// Types/States/MurrIOMOdule/MOM_STATES
{attribute 'strict'}
{attribute 'qualified_only'}
TYPE MOM_STATES :
(
	Idle := 0,
	Reverse := 1,
	Reversing := 2,
	ReverseToPrinthead := 3,
	ReversingToPrintHead := 4,
	ReverseDone := 5,
	WaitingForPrinter := 10,
	FeedToPrintOffset := 11,
	FeedingToPrintOffset := 12,
	FedToPrintOffset := 13,
	FeedAtPrintSpeed := 20,
	FeedingAtPrintSpeed := 21,
	FedAtPrintSpeed := 22,
	FeedBagOut := 30,
	FeedingBagOut := 31,
	FedBagOut := 32,
	Ready := 40,
	FeedToEye := 50,
	FeedingToEye := 51,
	SetTorqueMode := 52,
	Fault := 99,
	Manual := 100
);
END_TYPE

// Types/States/JOG_STATES
{attribute 'strict'}
{attribute 'qualified_only'}
TYPE JOG_STATES :
(
    Idle := 0,
    JogForwardDIRequest := 10,
    JogForwardOpcodeRequest := 11,
    JoggingForward := 12,
    JogReverseDIRequest := 20,
    JogReverseOpcodeRequest := 21,
    JoggingReverse := 22,
    StoppingJog := 30
);
END_TYPE

// Types/Fault
TYPE Fault :
STRUCT
    name : STRING[20];
    description : STRING[255];
END_STRUCT
END_TYPE

// Types/QX_PROGRAMS
{attribute 'strict'}
TYPE QX_PROGRAMS :
(
    HOME_HARD_STOP := 1
);
END_TYPE

// Types/Factoy Selection/ExteralConveyorSelection
{attribute 'qualified_only'}
{attribute 'strict'}
TYPE ExteralConveyorSelection :
(
	NotInstalled := 0,
	ExternalExitConveyor := 1
);
END_TYPE

// Types/PRINT_SPEEDS
{attribute 'qualified_only'}
{attribute 'strict'}
TYPE PRINT_SPEEDS :
(
	Two_IPS := 2
);
END_TYPE

// Types/States/PRESSURE_BAR_STATES
{attribute 'strict'}
{attribute 'qualified_only'}
TYPE PRESSURE_BAR_STATES :
(
	Idle := 0,
	OpenJaw := 10,
	OpeningJaw := 11,
	JawOpened := 12,
	CloseJaw := 20,
	ClosingJaw := 21,
	JawClosed := 22,
	Sealing := 30,
	Manual := 40,
	Homing := 41,
	Fault := 99
);
END_TYPE

// Types/Factoy Selection/BCVSelection
{attribute 'qualified_only'}
{attribute 'strict'}
TYPE BCVSelection :
(
	NotInstalled := 0,
	VisionBased := 1,
	LaserScanner := 2,
	TwoDimensional := 3
);
END_TYPE

// Types/States/MurrIOMOdule/MURR_SYSTEM_STATES
{attribute 'qualified_only'}
TYPE MURR_SYSTEM_STATES :
(
	Internal_Comm_OK := 1,
	Waiting_For_MOM := 2,
	Configuring_MOM := 4,
	Internal_Comm_Disabled := 8,
	No_Comm_To_Configured_Node := 127
);
END_TYPE

// Types/States/Head/HEAD_STATES
{attribute 'qualified_only'}
{attribute 'strict'}
TYPE HEAD_STATES :
(
	Idle := 0,
	SealAndSeparateBag := 10,
	SealingAndSeparatingBag := 11,
	SealedAndSeparatedBag := 12,
	ReleaseAndFeedBag := 20,
	ReleasingAndFeedingBag := 21,
	ReleasedAndFedBag := 22,
	OpenBag := 30,
	OpeningBag := 31,
	OpenedBag := 32,
	FinishCycle := 40, 
	FinishingCycle := 41,
	FinishedCycle := 42,
	StartReset := 50,
	Resetting := 51,
	StartHoming := 53,
	Homing := 54,
	HomingComplete := 55,
	MovePassthrough := 60,
	MovingPassthrough := 61,
	MovedPassthrough := 62,
	Fault := 99
);
END_TYPE

// Types/States/Head/SEAL_FLATTENER_STATES
{attribute 'strict'}
{attribute 'qualified_only'}
TYPE SEAL_FLATTENER_STATES :
(
	Idle := 0,
	MoveFlattenersOut := 10,
	MovingFlattenersOut := 11,
	MovedFlattenersOut := 12,
	MoveFlattenersUpAndToClearance := 20,
	MovingFlattenersUpAndToClearance := 21,
	MovedFlattenersUpAndToClearance := 22,
	MoveFlattenersToBagFeed := 23,
	MovingFlattenersToBagFeed := 24,
	MovedFlattenersToBagFeed := 25,
	MoveFlattenersIn := 30,
	MovingFlattenersIn := 31,
	MovedFlattenersIn := 32,
	MoveFlattenersDown := 40,
	MovingFlattenersDown := 41,
	MovedFlattenersDown := 42,
	MoveFlattenersToBagHolding := 50,
	MovingFlattenersToBagHolding := 51,
	MovedFlattenersToBagHolding := 52,
	Ready := 60,
	Fault := 99
);
END_TYPE

// Types/Factoy Selection/BagDeflatorSelection
{attribute 'qualified_only'}
{attribute 'strict'}
TYPE BagDeflatorSelection :
(
	NotInstalled := 0,
	IBDStandard := 1,
	IBDWithHingedPlate := 2,
	MotorizedIBD := 3
);
END_TYPE

// Types/States/Head/SEAL_BAR_STATES
{attribute 'strict'}
{attribute 'qualified_only'}
TYPE SEAL_BAR_STATES :
(
	Idle := 0,
	ExtendSealBar := 10,
	ExtendingSealBar := 11,
	SealBarExtened := 12,
	RetractSealBar := 20,
	RetractingSealBar := 21,
	RetractedSealBar := 22,
	Fault := 99
);
END_TYPE

// Types/States/Head/SEAL_SEPARATE_STATES
{attribute 'qualified_only'}
{attribute 'strict'}
TYPE SEAL_SEPARATE_STATES :
(
	Idle := 0,
	BringInIBD := 8,
	WaitForJawCloseDelay := 9,
	MoveJawIn := 10,
	MovingJawIn := 11,
	MovedJawIn := 12,
	ReverseBag := 20,
	ReversingBag := 21,
	ReversedBag := 22,
	SealBag := 30, 
	SealingBag := 31, 
	SealedBag := 32,
	Done := 100,
	Fault := 99
);
END_TYPE

// Types/ServiceCommands
TYPE ServiceCommands : 
STRUCT
	extendCommand : BOOL;
	retractCommand : BOOL;
	exhaustCommand : BOOL;
	extendedFeedback : BOOL;
	retractedFeedback : BOOL;
END_STRUCT
END_TYPE

// Types/States/VACUUM_PICKER_STATES
{attribute 'strict'}
{attribute 'qualified_only'}
TYPE VACUUM_PICKER_STATES :
(
	Idle := 0,
	Home := 1, 
	Homing := 2, 
	Homed := 3,
	XAxisMoveIn := 10,
	XAxisMovingIn := 11, 
	XaxisMovedIn := 12,
	VacuumTurnOn := 20,
	VacuumHeadDown := 30,
	YAxisMoveDown := 31,
	VacuumHeadAndYAxisMovingDown := 32,
	VacuumHeadAndYAxisMovedDown := 33,
	VacuumTurnOff := 40,
	ConveyorTurnOn := 50,
	ConveyorMoving := 51,
	ConveyorDone := 52,

	Fault := 99,
	Ready := 100,
	Manual := 101
);
END_TYPE

// FBs/Components/FB_MotorizedIBD/MotorizedIBDStates
{attribute 'qualified_only'}
{attribute 'strict'}
TYPE MotorizedIBDStates :
(
	Idle := 0,
	Homing := 9,
	Initialize := 10,
	Initializing := 11,
	Initialized := 12,
	MoveJawOut := 20,
	MovingJawOut := 21,
	MovedJawOut := 22,
	MoveJawIn := 30,
	MovingJawIn := 31,
	MovedJawIn := 32,
	StartClamping := 40,
	StartedClamping := 41,
	Clamping := 42, 
	ReleaseClamp := 43, 
	ReleasingClamp := 44,
	MoveOutFull := 50,
	MovingOutFull := 51,
	MovedOutFull := 52,
	Faulting := 98,
	Faulted := 99
);
END_TYPE

// FBs/Components/DelayDwellFB/DELAY_DWELL_STATES
{attribute 'qualified_only'}
{attribute 'strict'}
TYPE DELAY_DWELL_STATES :
(
	Idle := 0,
	Delay := 1,
	Dwell := 2,
	ResettingDwell := 10,
	ManualOn := 20,
	ManualOff := 21
);
END_TYPE

// Types/Factoy Selection/SealFlattenerSelection
{attribute 'qualified_only'}
{attribute 'strict'}
TYPE SealFlattenerSelection :
(
	NotInstalled := 0,
	MotorizedSealFlatteners := 1
);
END_TYPE

// Types/States/OPCODE_MODBUS_COMMAND_STATES
{attribute 'strict'}
{attribute 'qualified_only'}
TYPE OPCODE_MODBUS_COMMAND_STATES :
(
	Idle := 0,
	SendOpcodeAndParameters := 10,
	WaitAfterOpcodeAndParametersSent := 11,
	Fault := 99
);
END_TYPE

// Types/States/FILLER_STATES
{attribute 'strict'}
{attribute 'qualified_only'}
TYPE FILLER_STATES :
(
	Idle := 0,
	CycleBaggerToActiveFiller := 10,
	WaitingForFiller := 11,
	Dropping := 13,
	BaggerCycling := 14,
	Fault := 99
);
END_TYPE

// Types/States/Head/FINISH_CYCLE_STATES
{attribute 'qualified_only'}
{attribute 'strict'}
TYPE FINISH_CYCLE_STATES :
(
	Idle := 0,
	Start := 1,
	OpenFunnel := 10, 
	OpeningFunnel := 11, 
	OpenedFunnel := 12,
	ClosingFunnelForRetry := 13,
	FunnelClosed := 14,
	BringSealFlattenersInAndDown := 20, 
	BringingSealFlattenersInAndDown := 21,
	SealFlattenersInAndDown := 22,
	BringSealFlattenersToBagHolding := 30,
	BringingSealFlattenersToBagHolding := 31,
	SealFlattenersAtBagHolding := 32,
	Done := 100,
	Fault := 99
);
END_TYPE

// Types/States/GRABBER_STATES
{attribute 'strict'}
{attribute 'qualified_only'}
TYPE GRABBER_STATES :
(
	Idle := 0,
	OpenGrippers := 10,
	MoveGrippersOut := 11,
	MovingGrippersOut := 12,
	GrippersMovedOut :=13,
	MoveGantryUp := 20,
	MovingGantryUp := 21,
	GantryMovedUp := 22,
	MoveGrippersIn := 30,
	MovingGrippersIn := 31,
	GrippersMovedIn := 32,
	Ready := 40,
	GrabBag := 50,
	MoveGantryDown := 60,
	MovingGantryDown := 61,
	GantryMovedDown := 62,
	ReleaseBag := 70,
	Fault := 99
);
END_TYPE

// Types/Factoy Selection/PalmButtonSelection
{attribute 'qualified_only'}
{attribute 'strict'}
TYPE PalmButtonSelection :
(
	NotInstalled := 0,
	SinglePalmButton := 1,
	DualPalmButton := 2,
	LightedPalmButton := 3
);
END_TYPE

// FBs/Fault/LogMessageType
TYPE LogMessageType :
STRUCT
	logTime : DATE_AND_TIME;
	logMessage : STRING;
END_STRUCT
END_TYPE

// Types/ORIENTAL_OPERATION_TYPES
{attribute 'qualified_only'}
{attribute 'strict'}
TYPE ORIENTAL_OPERATION_TYPES :
(
    NoSetting := 0,
    AbsolutePositioning := 1,
    IncrementalPositioning := 2
);
END_TYPE

// FBs/Components/KeyenceL20FB/eKeyenceLN20_Error_ID
{attribute 'qualified_only'}
{attribute 'strict'}
TYPE eKeyenceLN20_Error_ID :
(
	NO_ERROR := 0,
	OPERATION_INSTRUCTION_ERROR := 120,
	BANK_NUMBER_ERROR := 102,
	EIP_UPDATE_ERROR := 230
);
END_TYPE

// FBs/Components/FB_MotorizedPressureBar/MotorizedPbarStates
{attribute 'qualified_only'}
{attribute 'strict'}
TYPE MotorizedPbarStates :
(
	Idle := 0,
	Homing := 9,
	Initialize := 10,
	Initializing := 11,
	Initialized := 12,
	MoveJawOut := 20,
	MovingJawOut := 21,
	MovedJawOut := 22,
	MoveJawIn := 30,
	MovingJawIn := 31,
	MovedJawIn := 32,
	StartClamping := 40,
	StartedClamping := 41,
	Clamping := 42, 
	ReleaseClamp := 43, 
	ReleasingClamp := 44,
	Faulting := 98,
	Faulted := 99
);
END_TYPE

// Types/States/BCR_STATES
{attribute 'strict'}
{attribute 'qualified_only'}
TYPE BCR_STATES :
(
	Idle := 0,
	WaitForOffset := 10,
	TriggerReader := 11,
	WaitingForResult := 12,
	Resetting := 13
);
END_TYPE

// Types/PressureBarFaultsType
TYPE PressureBarFaultsType :
STRUCT
	failedToOpen : FB_Fault(name := 'Pressure Bar Failed to Open');        // Pressure Bar was commanded to extend but failed to reach the sensor
    failedToClose : FB_Fault(name := 'Pressure Bar Failed to Close');      // Pressure Bar was commanded to retract but failed to reach the sensor
	sensorFault : FB_Fault(name := 'Pressure Bar Sensor Fault');		// Both the open and close sensors active at the same time
	obstructionDetected : FB_Fault(name := 'Pressure Bar Obstruction Detected');		// Pressure Bar detected an obstruction
	obstructionFailedToSwitch : FB_Fault(name := 'Pressure Bar Obstruction Detected'); // Pressure bar obstruction sensors should switch when closed
END_STRUCT
END_TYPE

// Types/Factoy Selection/BagOpenFingersSelection
{attribute 'qualified_only'}
{attribute 'strict'}
TYPE BagOpenFingersSelection :
(
	NotInstalled := 0,
	PneumaticWithBagOpenSensors := 1
);
END_TYPE

// Types/HMI Types/PressureBarHMI
TYPE PressureBarHMI :
STRUCT
	openDelay : UINT;
	closeDelay : UINT;
	passthroughSetting : REAL;
	lowPressureAirDwell : REAL;
	highPressureAirDwell : REAL;
END_STRUCT
END_TYPE

// Types/AuxIO/AuxInputSelection
{attribute 'qualified_only'}
{attribute 'strict'}
TYPE AuxInputSelection :
(
	NotConfigured := 0,
	BaggerInhibit := 1
);
END_TYPE

// Types/States/PRINT_AND_APPLY_STATES
{attribute 'strict'}
{attribute 'qualified_only'}
TYPE PRINT_AND_APPLY_STATES :
(
	Idle := 0,
	WaitForLabel := 10,
	WaitForLOTAR := 11,
	ReadyToApply := 12,
	Applying := 13, 
	Fault := 99
);
END_TYPE

// Types/States/Head/RELEASE_FEED_STATES
{attribute 'qualified_only'}
{attribute 'strict'}
TYPE RELEASE_FEED_STATES :
(
	Idle := 0,
	MoveJawOutAndDropBag := 10,
	MovingJawOutAndDroppingBag := 11,
	MovingJawOutAndFeedBag := 12,
	MovingJawOutAndFeedingBag := 13,
	MovedJawOutAndFedBag := 15,
	WaitForPrinter := 20,
	FeedToOffset := 21,
	FeedingToOffset := 22,
	StartPrinting := 23,
	SendPrintSignal := 24,
	Printing := 25, 
	StopPrinting := 26,
	Done := 100,
	Fault := 99
);
END_TYPE

// Types/IOMasterFaultsType
TYPE IOMasterFaultsType :
STRUCT
	commFail : FB_Fault(name := 'Communication Fail');	// IO Master to Controller Communication Failure
END_STRUCT
END_TYPE

// Types/CylinderFaultsType
TYPE CylinderFaultsType :
STRUCT
	failedToExtend : FaultType;        // Cylinder was commanded to extend but failed to reach the sensor
    failedToRetract : FaultType;      // Cylinder was commanded to retract but failed to reach the sensor
	sensorFault : FaultType;		// Both Extend and Retract sensors active at the same time
END_STRUCT
END_TYPE

// Types/States/EZFEED_STATES_1
{attribute 'strict'}
{attribute 'qualified_only'}
TYPE EZFEED_STATES_1 :
(
	Idle := 0,
	IndexingFlightMode := 10,
	IndexingPartsMode := 11,
	IndexDwell := 12,
	WaitForBaggerCycleComplete := 13,
	PartsStarved := 20,
	Fault := 99
);
END_TYPE

// Types/ModbusLongType
TYPE ModbusLongType :
STRUCT
    highWord : WORD;
    lowWord : WORD;
    displayValue : DINT;
    rawValue : DINT;
END_STRUCT
END_TYPE

// Types/Alarm
TYPE Alarm :
STRUCT
	active : BOOL;
	acknowledged : BOOL;
	ackCommand : BOOL;
END_STRUCT
END_TYPE

// Types/Factoy Selection/AuxiliaryIOSelection
{attribute 'qualified_only'}
{attribute 'strict'}
TYPE AuxiliaryIOSelection :
(
	NotInstalled := 0,
	AuxIOStandard := 1
);
END_TYPE

// Types/States/PASSTHROUGH_SERVO_STATES
{attribute 'strict'}
{attribute 'qualified_only'}
TYPE PASSTHROUGH_SERVO_STATES :
(
	Idle := 0,
	HomingRequired := 1,
	StartHoming := 10,
	Homing := 11,
	HomeComplete := 12,
	MovePassthroughOut := 20,
	MovingPassthroughOut := 21,
	PassthroughMovedOut := 22,
	MovePassthroughIn := 30,
	MovingPassthroughIn := 31,
	PassthroughMovedIn := 32,
	Ready := 40,
	Fault := 99
);
END_TYPE

// Types/States/Head/BAG_DELIVERY_STATES
{attribute 'strict'}
{attribute 'qualified_only'}
TYPE BAG_DELIVERY_STATES :
(
	Idle := 0,
	Reverse := 1,
	Reversing := 2,
	ReverseToPrinthead := 3,
	ReversingToPrintHead := 4,
	ReverseDone := 5,
	WaitingForPrinter := 10,
	FeedToPrintOffset := 11,
	FeedingToPrintOffset := 12,
	FedToPrintOffset := 13,
	FeedAtPrintSpeed := 20,
	FeedingAtPrintSpeed := 21,
	FedAtPrintSpeed := 22,
	FeedBagOut := 30,
	FeedingBagOut := 31,
	FedBagOut := 32,
	Ready := 40,
	FeedToEye := 50,
	FeedingToEye := 51,
	SetTorqueMode := 52,
	Fault := 99,
	Manual := 100
);
END_TYPE

// Types/AuxIO/AuxIOConfiguration
TYPE AuxIOConfiguration :
STRUCT
	factorySelection : AuxiliaryIOSelection;
	cfgInputSelection : AuxInputSelection;
	cfgOutput1Selection : AuxOutputSelection;
	cfgOutput2Selection : AuxOutputSelection;
END_STRUCT
END_TYPE

// Types/FaultType
TYPE FaultType :
STRUCT
	active : BOOL;
	acknowledged : BOOL;
	ackCommand : BOOL;
END_STRUCT
END_TYPE

// FBs/Components/KeyenceL20FB/eKeyenceLN20FB_States
{attribute 'qualified_only'}
{attribute 'strict'}
TYPE eKeyenceLN20FB_States :
(
	Idle := 0,
	WaitForStatus := 2,
	SetStatus := 3,
	WaitForReadClear := 4,
	Reset := 100
);
END_TYPE

// Types/Warning
TYPE Warning :
STRUCT
	active : BOOL;
END_STRUCT
END_TYPE

// Types/StepServoFaultsType
TYPE StepServoFaultsType :
STRUCT
	positionLimit : FB_Fault(name := 'Motor exceeded position limit - following error');        // Motor exceeded position limit - following error
	CCWLimit : FB_Fault(name := 'Counter-Clockwise Limit Reached'); // Counter-Clockwise Limit Reached
	CWLimit : FB_Fault(name := 'Clockwise Limit Reached');		// Clockwise Limit Reached
    overTemp : FB_Fault(name := 'Motor Over Temperature Limit');      // Motor Over Temperature Limit
    internalVoltage : FB_Fault(name := 'Internal Voltage Fault');      // Internal Voltage Fault
    overVoltage    : FB_Fault(name := 'Overvoltage Fault');      // Overvoltage Fault
	underVoltage : FB_Fault(name := 'Undervoltage Fault'); 	// Undervoltage Fault
    overCurrent : FB_Fault(name := 'Motor Overcurrent');      // Motor Overcurrent
    openMotorWinding : FB_Fault(name := 'Motor Detected Open Winding');      // Motor Detected Open Winding
    badEncoder : FB_Fault(name := 'Motor Encoder Failure');      // Motor Encoder Failure
	noMove : FB_Fault(name := 'No Move After Command');
	currentFoldback : FB_Fault(name := 'Current Foldback');
	commFail : FB_Fault(name := 'Drive to Controller Communication Failure');	// Drive to Controller Communication Failure
	notHomed : FB_Fault(name := 'Drive is not homed'); // Drive is not homed
END_STRUCT
END_TYPE

// Types/Factoy Selection/FillerSelection
{attribute 'qualified_only'}
{attribute 'strict'}
TYPE FillerSelection :
(
	NotInstalled := 0,
	StandardFiller := 1,
	EZFeed := 2
);
END_TYPE

// Types/Factoy Selection/ModelSelection
{attribute 'qualified_only'}
{attribute 'strict'}
TYPE ModelSelection :
(
	Pro18 := 0,
	Pro24 := 1,
	Pro18_02 := 2
);
END_TYPE

// Types/STEP_SERVO_OPCODES
{attribute 'strict'}
{attribute 'qualified_only'}
//Taken from Host-Command-Reference pdf on Applied Motion website
TYPE STEP_SERVO_OPCODES :
(
	ALARM_RESET := 16#BA,     
	START_JOGGING := 16#96,     
	STOP_JOGGING := 16#D8,     
	ENCODER_FUNCTION := 16#D6,     //0
	ENCODER_POSITION := 16#98,     //Position
	FEED_TO_DOUBLE_SENSOR := 16#69,     //I/O Point 1 Condition 1 I/O Point 2 Condition 2
	FOLLOW_ENCODER := 16#CC,     //I/O Point Condition
	FEED_TO_LENGTH := 16#66,     
	FEED_TO_SENSOR_WITH_MASK_DISTANCE := 16#6A,     //I/O Point Condition
	FEED_AND_SET_OUTPUT := 16#68,     //I/O Point Condition
	FEED_TO_POSITION := 16#67,     
	FEED_TO_SENSOR := 16#6B,     //I/O Point Condition
	FEED_TO_SENSOR_WITH_SAFETY_DISTANCE := 16#6C,     //I/O Point Condition
	JOG_DISABLE := 16#A3,     
	JOG_ENABLE := 16#A2,     
	MOTOR_DISABLE := 16#9E,     
	MOTOR_ENABLE := 16#9F,     
	SEEK_HOME := 16#6E,     //I/O Point Condition
	SET_POSITION := 16#A5,     //Position
	FILTER_INPUT := 16#C0,     //I/O Point Filter Time
	FILTER_SELECT_INPUTS := 16#D3,     
	STEP_FILTER_FREQ := 16#06,     //Freq
	ANALOG_DEADBAND := 16#D2,     //0.001 V
	ALARM_RESET_INPUT := 16#46,     //Function ('1'..'3') I/O Point
	ALARM_OUTPUT := 16#47,     //Function ('1'..'3') I/O Point
	ANALOG_SCALING := 16#D1,     
	DEFINE_LIMITS := 16#42,     //1..3
	SET_OUTPUT := 16#8B,     //I/O Point Condition
	WAIT_FOR_INPUT := 16#70,     
	QUEUE_LOAD_AND_EXECUTE := 16#78,     //1..12
	WAIT_TIME := 16#6F,     //0.01 sec
	STOP_MOVE_KILL_BUFFER := 16#E1,    
	STOP_MOVE_KILL_BUFFER_NORMAL_DECEL := 16#E2,
	STOP_MOVE := 16#B5  // Might work, might not     
);
END_TYPE

// Types/Factoy Selection/FunnelSelection
{attribute 'qualified_only'}
{attribute 'strict'}
TYPE FunnelSelection :
(
	NotInstalled := 0,
	FunnelWithSensors := 1,
	FunnelWithoutSensors := 2
);
END_TYPE

// Types/CONFIG_VERSIONS
{attribute 'strict'}
{attribute 'qualified_only'}
TYPE CONFIG_VERSIONS :
(
	V_1_0,
	V_1_1,
	V_1_2,
	V_1_3,
	V_1_4,
	V_1_5,
	V_1_6,
	V_1_7,
	V_1_8,
	V_1_9,
	V_1_10,
	V_1_11,
	V_1_12,
	V_1_13,
	V_1_14,
	V_1_15,
	V_1_16,
	V_1_17,
	V_1_18,
	V_1_19,
	V_1_20,
	V_1_21,
	V_1_22,
	V_1_23,
	V_1_24,
	V_1_25,
	V_1_26,
	V_1_27,
	V_1_28,
	V_1_29,
	V_1_30,
	V_1_31,
	V_1_32,
	V_1_33,
	V_1_34,
	V_1_35,
	V_1_36,
	V_1_37,
	V_1_38,
	V_1_39,
	V_1_40,
	V_1_41,
	V_1_42,
	V_1_43,
	V_1_44,
	V_1_45,
	V_1_46,
	V_1_47,
	V_1_48,
	V_1_49,
	V_2_0,
	V_2_1,
	V_2_2,
	V_2_3,
	V_2_4,
	V_2_5,
	V_2_6,
	V_2_7,
	V_2_8,
	V_2_9,
	V_2_10,
	V_2_11,
	V_2_12,
	V_2_13,
	V_2_14,
	V_2_15,
	V_2_16,
	V_2_17,
	V_2_18,
	V_2_19,
	V_2_20,
	V_2_21,
	V_2_22,
	V_2_23,
	V_2_24,
	V_2_25,
	V_2_26,
	V_2_27,
	V_2_28,
	V_2_29,
	V_2_30,
	V_2_31,
	V_2_32,
	V_2_33,
	V_2_34,
	V_2_35,
	V_2_36,
	V_2_37,
	V_2_38,
	V_2_39,
	V_2_40,
	V_2_41,
	V_2_42,
	V_2_43,
	V_2_44,
	V_2_45,
	V_2_46,
	V_2_47,
	V_2_48,
	V_2_49
);
END_TYPE

// Types/States/JAW_HOMING_STATES
{attribute 'strict'}
{attribute 'qualified_only'}
TYPE JAW_HOMING_STATES :
(
    Idle := 0,
    MoveForwardFromSensor := 10,
    MovingForwardFromSensor := 11,
	ClearToHome := 12,
    StartHoming := 13,
    Homing := 14,
    HomeComplete := 15,
	MoveToTwoInches := 16, 
	MovingToTwoInches := 17,
	SetLimits := 18
	
);
END_TYPE

// FBs/Components/EZFeedFB/EZFEED_STATES
{attribute 'strict'}
{attribute 'qualified_only'}
TYPE EZFEED_STATES :
(
	Idle := 0,
	IndexingFlightMode := 10,
	IndexingPartsMode := 11,
	IndexDwell := 12,
	WaitForBaggerCycleComplete := 13,
	PartsStarved := 20,
	Fault := 99
);
END_TYPE

// Types/States/Head/BAG_OPEN_ASSIST_STATES
{attribute 'qualified_only'}
{attribute 'strict'}
TYPE BAG_OPEN_ASSIST_STATES :
(
	Idle := 0,
	MoveJawIn := 10,
	MovingJawIn := 11,
	MovedJawIn := 12,
	MoveJawOut := 20,
	MovingJawOutAndGrab := 21,
	CheckForSuccessfulBagGrab := 22,
	BagFailedToOpen := 23,
	BagOpened := 24,
	MovingJawOutAfterGrab := 25,
	MovedJawOut := 26,
	FeedNewBag := 27,
	Done := 100,
	Fault := 99
);
END_TYPE

// ElectricMachine/Application/HMIData
// All HMI data is presented through this GVL
{attribute 'qualified_only'}
{attribute 'global_init_slot' := '50001'}
VAR_GLOBAL //PERSISTENT RETAIN
	initiateCycle : BOOL;  // Initiate Cycle Pushbutton
	ackAllFaults : BOOL; // Acknowledge All Faults from HMI
	makeReady : BOOL;
	jobLoaded : BOOL;
    stopMachine : BOOL;
	version : STRING;
	inCycle : BOOL;
	batchEnable : BOOL;
	autoEnable : BOOL;
	autoDwell : REAL;
	batchSetting : UDINT := 10;
	batchCount : UDINT;
	headCycleCount : UDINT;
	pressureBarOpenDelay : REAL;
	pressureBarCloseDelay : REAL;
	passthroughSetting : REAL := 5.0;
	passthroughOffset : REAL;
	passthroughPosition : REAL;
	lpaDwell : REAL;
	hpaDwell : REAL;
	sealBarDwell : REAL;
	sealBarTemperatureSetting : UDINT;
	sealBarTemperature : UDINT;
	sealFlattenersPosition : REAL;
	bagSkirtLength : REAL := 1.35;
	bagLength : REAL := 23.5;
	bagWidth : REAL := 17.5;
	bagThickness : REAL := 2.5;
	bagTensionSetting : REAL := 0.6;  // Bag takeup tension setting in amps
	bagDropTime : REAL;
	bagForwardSpeed : UDINT := 55;
	bagReverseSpeed : UDINT := 3;
	bagEdgePhotoeyeCovered : BOOL;
	printSpeed : UDINT := 6;
	printLength : REAL := 8.0;
	printOffset : REAL := 2.0;
	fillerCountSetting : UDINT;
	fillerCurrentCount : UDINT;
	fillerDropTime : REAL;
	fillerEnable : BOOL;
	loadPlateDelay : REAL;
	loadPlateDwell : REAL;
	exitConveyorDwell : REAL;
	vacuumDwell : REAL := 0.25;
	IBDDeflateDwellTime  : REAL := 0.75;
	IBDPackageEjectAssistDelayTime : REAL;
	IBDPackageEjectAssistDwellTime : REAL := 0.8;
	funnelInUse : BOOL;								// Funnel Enable/Disable
	funnelOpenDelay : REAL := 0.25;					// Funnel Open Delay after pressure bar open
	funnelOpeningTime : REAL := 0.5;				// For funnel w/o sensors only : Time required to consider funnel open after command to open
	funnelClosingTime : REAL := 0.5;				// For funnel w/o sensors only : Time required to consider funnel closed after command to close
	externalExitConveyorDwell : REAL;
	barcodeGoodReadCount : UDINT;
	barcodeBadReadCount : UDINT;
	barcodeBadReadFaultSetting : UDINT;
	barcodeStartPosition : REAL;
	barcodeScanDistance : REAL := 1.0;
	barcodeVerifierInUse : BOOL;
	barcodeLastReadString : STRING[100];
	lastCycleTime : REAL;
	averageCycleTime : REAL;
	resetAverageCycleTime : BOOL;
	bagOpenRetrySetting : INT := 3;
	bagOpenRetryCount : INT;
	bagOpenFeedNewBagSetting : INT := 1;
	bagOpenFeedNewBagCount : INT;
	currentJobID : INT;
	separateBeforeSeal : BOOL;
	activateDemoMode : BOOL;
	printerInUse : BOOL;
	printerInstalled : BOOL;
	lpaDuringBagFeedEnable : BOOL := TRUE;
	lpaBagEjectAssistEnable : BOOL := TRUE;
	infeedConveyorRunningMode : BOOL;  			//0 = Indexing, 1 = Continuous
	infeedConveyorCountingMode : BOOL;			// 0 = Flight, 1 = Parts
	infeedIndexDwellTimer : REAL := 0.25;
	infeedFlightCountTarget : DINT := 5;
	infeedFlightCountActual : DINT;
	infeedPartsCountTarget : DINT := 10;
	infeedPartsCountActual : DINT;
	infeedEmptyPartsSetting : DINT := 10;
	infeedEmptyPartsActual : DINT;
	printAndApplyConveyorDwell : REAL := 5.0;
	printAndApplyProductToPhotoeyeTime : REAL := 4.0;
	printAndApplyWaitForLabelTimeout : REAL := 15.0;
	
	(*Service Stuff*)
	lpaServiceOn : BOOL;
	lpaServiceOff : BOOL;
	lpaServicePulse : BOOL;
	hpaServiceOn :BOOL;
	hpaServicePulse : BOOL;
	exitConveyorStart : BOOL;
	exitConveyorStop : BOOL;
	exitConveyorJog : BOOL;
	exitConveyorJogTime : TIME;
	exitConveyorStartDwell : BOOL;
	pressureBarService : ServiceCommands;
	loadPlateService : ServiceCommands;
	forwardLoadPlateService : ServiceCommands;
	rearLoadPlateService : ServiceCommands;
	loadShelfService : ServiceCommands;
	IBDService : ServiceCommands;
	funnelService : ServiceCommands;
	baggerHeadService : ServiceCommands;
	jogBagForward : BOOL;
	jogBagReverse : BOOL;
	jogPassthroughForward : BOOL;
	jogPassthroughReverse : BOOL;
	sealBarServiceCycle : BOOL;
	sealBarServiceRetract : BOOL;
	sealBarServiceExtend : BOOL;
	bagOpenFingersServiceGrab : BOOL;
	bagOpenFingersServiceRelease : BOOL;
	sealFlattenersServiceRaise : BOOL;
	sealFlattenersServiceLower : BOOL;
	sealFlattenersServiceJogIn : BOOL;
	sealFlattenersServiceJogOut : BOOL;
	sealFlattenersManualPositionSetting : REAL;
	sealFlattenersMoveToManualPos : BOOL;
	passthroughManualPositionSetting : REAL;
	passthroughMoveToManualPos : BOOL;
	factoryTestMode : BOOL;
	vacuumServiceOn : BOOL;
	vacuumServiceOff : BOOL;
	printHeadServiceRaise : BOOL;
	printHeadServiceLower : BOOL;
	externalExitConveyorStart : BOOL;
	externalExitConveyorStop : BOOL;
	externalExitConveyorJog : BOOL;
	externalExitConveyorStartDwell : BOOL;
	triggerBarcodeReaderService : BOOL;
	IBDOffset : REAL := 3.0;
	
	(*Factoy Config*)
	bofSelection : BagOpenFingersSelection := BagOpenFingersSelection.PneumaticWithBagOpenSensors;
	sealFlattenersSelection : SealFlattenerSelection := SealFlattenerSelection.MotorizedSealFlatteners;
	printerSelection : LabelPrinterSelection := LabelPrinterSelection.ZebraPrinter203DPI;
	integratedExitConveyorSelection : IntegratedConveyorSelection := IntegratedConveyorSelection.RearExit;
	externalExitConveyorSelection : ExteralConveyorSelection := ExteralConveyorSelection.NotInstalled;
	packageEjectSelection : PackageEjectionSelection := PackageEjectionSelection.RearRetractingLoadPlate;
	independentBagDeflatorSelection : BagDeflatorSelection := BagDeflatorSelection.NotInstalled;
	cycleStartButtonSelection : PalmButtonSelection := PalmButtonSelection.DualPalmButton;
	barcodeVerifierSelection : BCVSelection := BCVSelection.NotInstalled;
	baggerModelSelection : ModelSelection;
	auxIOConfig : AuxIOConfiguration;
	fillerFactorySelection : FillerSelection;
	funnelFactorySelection : FunnelSelection;
	murrIOConfigVersion : CONFIG_VERSIONS := CONFIG_VERSIONS.V_1_4;
	printerConfigVersion : CONFIG_VERSIONS := CONFIG_VERSIONS.V_1_2;
	frontFilmFeedMotorConfigVersion : CONFIG_VERSIONS := CONFIG_VERSIONS.V_1_0;
	rearUnwindMotorConfigVersion : CONFIG_VERSIONS := CONFIG_VERSIONS.V_1_1;
	sealFlattenerMotorConfigVersion : CONFIG_VERSIONS := CONFIG_VERSIONS.V_1_0;
	
	(*Warnings*)
	printerRibbonLow : Warning;
	printerNotReady : Warning;
	waitingForPrinter : Warning;
	sealBarNotAtTemperature : Warning;
	recoveryModeActive : Warning;
	jobLoadRequired : Warning;
	baggerNotReady : Warning;
	demoModeIsActive : Warning;
	factoryTestModeActive : Warning;
	machineNotTested : Warning;
	packageEjectGuardRemoved : Warning;
	bagLevelLow : Warning;
	fillerModeCycleStartOnly : Warning;
	baggerInhibited : Warning;
	infeedConveyorOutOfParts : Warning;
	mayCycleUnexpectedly : Warning;
	printAndApplyRibbonLow : Warning;
	printAndApplyWaitingForApply : Warning;
	printAndApplyWaitingForLabel : Warning;
	printAndApplyBypassed : Warning;
	(*Misc*)
	pressureBarState : STRING;
    
    (*Counters*)
    baggerCycles : FB_CycleCounter;
	bagOpenFingerCycles : FB_CycleCounter;
	bagsMade : FB_CycleCounter;
	sealBarCycles : FB_CycleCounter;
	pressureBarCycles : FB_CycleCounter;
	passthroughChanges : FB_CycleCounter;
	loadPlateCycles : FB_CycleCounter;
	printerCycles : FB_CycleCounter;
	motorizedSealFlattenerCycles : FB_CycleCounter;
	bagOpenRetryTotal : FB_CycleCounter;
	bagsRejectedTotal : FB_CycleCounter;
	resettableBagsMade : FB_CycleCounter;
	
	(*Predictive Maint.*)
	airFilterClean : FB_PredictiveMaint := (target := 30000, count := 0, name := 'Clean Air Filter');
	driveRollerClean : FB_PredictiveMaint := (target := 20000, count := 0, name := 'Clean Drive Rollers', units := 'Inches of Bag');
	printHeadClean : FB_PredictiveMaint := (target := 10000, count := 0, name := 'Clean Print Head', units := 'Printer Cycles');
	pressureBarGuideShaftGuides : FB_PredictiveMaint := (target := 0, count := 127888, name := 'Replace Guide Shafts');
	
	pressureBarLeak : FB_CylinderLeak := (maximumStrokeTime := 5.0, name := 'Pressure Bar Stroke', units := 'Seconds');
	loadPlateLeak : FB_CylinderLeak := (maximumStrokeTime := 2.0, name := 'Load Plate Stroke', units := 'Seconds');
	
	msfHorizontalMotorTemp : FB_DriveTemp := (maxTemp := 60.0, name := 'MSF Motor Temp.', units := 'deg C');
	bagDeliveryMotorTemp : FB_DriveTemp := (maxTemp := 60.0, name := 'Bag Delivery Motor Temp.', units := 'deg C');
	passthroughMotorTemp : FB_DriveTemp := (maxTemp := 60.0, name := 'Passthrough Motor Temp.', units := 'deg C');
	
	(*Info*)
	faultActive : BOOL;

END_VAR

VAR_GLOBAL CONSTANT
	murrIOConfigVersionMax : CONFIG_VERSIONS := CONFIG_VERSIONS.V_1_4;
	printerConfigVersionMax : CONFIG_VERSIONS := CONFIG_VERSIONS.V_1_2;
	frontFilmFeedMotorConfigVersionMax : CONFIG_VERSIONS := CONFIG_VERSIONS.V_1_0;
	rearUnwindMotorConfigVersionMax : CONFIG_VERSIONS := CONFIG_VERSIONS.V_1_1;
	sealFlattenerMotorConfigVersionMax : CONFIG_VERSIONS := CONFIG_VERSIONS.V_1_0;
END_VAR

// ObjectHandling/GlobalObjects
{attribute 'qualified_only'}
{attribute 'global_init_slot' := '49995'}
VAR_GLOBAL CONSTANT
	MAX_OBJECTS : UINT := 750;
	MAX_CYLINDERS : UINT := 20;
	MAX_MOTORS : UINT := 10;
	MAX_FAULTS : UINT := 300;
	MAX_LOGS : UINT := 100;
	MAX_LOGGABLE : UINT := 500;
	MAX_EXECUTEABLE : UINT := 300;
END_VAR

VAR_GLOBAL
	CollectionOfAllObjects : FB_CollectionHandlerAll; 
	CollectionOfFaults : FB_CollectionHandlerFaults; 
// 	CollectionOfCylinders : FB_CollectionHandlerCylinders;
// 	CollectionOfPositionableMotors : FB_CollectionHandlerPositionableMotors;
	CollectionOfActiveFaults : FB_CollectionHandlerActiveFaults; 
	CollectionOfLogs : FB_CollectionHandlerLogs; 
	CollectionOfLoggable : FB_CollectionHandlerLoggable;
	CollectionOfExecutable : FB_CollectionHandlerExecutable;
	CollectionOfInitialzable : FB_CollectionHandlerInitializable;
END_VAR

// Pro18_1174/Application/HMIData
// All HMI data is presented through this GVL
{attribute 'qualified_only'}
{attribute 'global_init_slot' := '50001'}
VAR_GLOBAL //PERSISTENT RETAIN
	initiateCycle : BOOL;  // Initiate Cycle Pushbutton
	ackAllFaults : BOOL; // Acknowledge All Faults from HMI
	makeReady : BOOL;
	jobLoaded : BOOL;
    stopMachine : BOOL;
	version : STRING;
	inCycle : BOOL;
	batchEnable : BOOL;
	batchSetting : UDINT := 10;
	batchCount : UDINT;
	headCycleCount : UDINT;
	pressureBarOpenDelay : REAL;
	pressureBarCloseDelay : REAL;
	passthroughSetting : REAL := 5.0;
	passthroughOffset : REAL;
	passthroughPosition : REAL;
	lpaDwell : REAL;
	hpaDwell : REAL;
	sealBarDwell : REAL;
	sealBarTemperatureSetting : UDINT;
	sealBarTemperature : UDINT;
	sealFlattenersPosition : REAL;
	bagSkirtLength : REAL := 1.35;
	bagLength : REAL := 23.5;
	bagWidth : REAL := 17.5;
	bagThickness : REAL := 2.5;
	bagTensionSetting : REAL := 0.6;  // Bag takeup tension setting in amps
	bagDropTime : REAL;
	bagForwardSpeed : UDINT := 55;
	bagReverseSpeed : UDINT := 3;
	bagEdgePhotoeyeCovered : BOOL;
	printSpeed : UDINT := 6;
	printLength : REAL := 8.0;
	printOffset : REAL := 2.0;
	fillerCountSetting : UDINT;
	fillerCurrentCount : UDINT;
	fillerDropTime : REAL;
	fillerEnable : BOOL;
	loadPlateDelay : REAL;
	loadPlateDwell : REAL;
	exitConveyorDwell : REAL;
	vacuumDwell : REAL := 0.25;
	IBDDeflateDwellTime  : REAL := 0.75;
	IBDPackageEjectAssistDelayTime : REAL;
	IBDPackageEjectAssistDwellTime : REAL := 0.8;
	funnelInUse : BOOL;								// Funnel Enable/Disable
	funnelOpenDelay : REAL := 0.25;					// Funnel Open Delay after pressure bar open
	funnelOpeningTime : REAL := 0.5;				// For funnel w/o sensors only : Time required to consider funnel open after command to open
	funnelClosingTime : REAL := 0.5;				// For funnel w/o sensors only : Time required to consider funnel closed after command to close
	externalExitConveyorDwell : REAL;
	barcodeGoodReadCount : UDINT;
	barcodeBadReadCount : UDINT;
	barcodeBadReadFaultSetting : UDINT;
	barcodeStartPosition : REAL;
	barcodeScanDistance : REAL := 1.0;
	barcodeVerifierInUse : BOOL;
	barcodeLastReadString : STRING[100];
	lastCycleTime : REAL;
	averageCycleTime : REAL;
	resetAverageCycleTime : BOOL;
	bagOpenRetrySetting : INT := 3;
	bagOpenRetryCount : INT;
	bagOpenFeedNewBagSetting : INT := 1;
	bagOpenFeedNewBagCount : INT;
	currentJobID : INT;
	separateBeforeSeal : BOOL;
	activateDemoMode : BOOL;
	printerInUse : BOOL;
	printerInstalled : BOOL;
	lpaDuringBagFeedEnable : BOOL := TRUE;
	lpaBagEjectAssistEnable : BOOL := TRUE;
	infeedConveyorRunningMode : BOOL;  			//0 = Indexing, 1 = Continuous
	infeedConveyorCountingMode : BOOL;			// 0 = Flight, 1 = Parts
	infeedIndexDwellTimer : REAL := 0.25;
	infeedFlightCountTarget : DINT := 5;
	infeedFlightCountActual : DINT;
	infeedPartsCountTarget : DINT := 10;
	infeedPartsCountActual : DINT;
	infeedEmptyPartsSetting : DINT := 10;
	infeedEmptyPartsActual : DINT;

	(*Service Stuff*)
	lpaServiceOn : BOOL;
	lpaServiceOff : BOOL;
	lpaServicePulse : BOOL;
	hpaServiceOn :BOOL;
	hpaServicePulse : BOOL;
	exitConveyorStart : BOOL;
	exitConveyorStop : BOOL;
	exitConveyorJog : BOOL;
	exitConveyorJogTime : TIME;
	exitConveyorStartDwell : BOOL;
	pressureBarService : ServiceCommands;
	loadPlateService : ServiceCommands;
	forwardLoadPlateService : ServiceCommands;
	rearLoadPlateService : ServiceCommands;
	loadShelfService : ServiceCommands;
	IBDService : ServiceCommands;
	funnelService : ServiceCommands;
	jogBagForward : BOOL;
	jogBagReverse : BOOL;
	jogPassthroughForward : BOOL;
	jogPassthroughReverse : BOOL;
	sealBarServiceCycle : BOOL;
	sealBarServiceRetract : BOOL;
	sealBarServiceExtend : BOOL;
	bagOpenFingersServiceGrab : BOOL;
	bagOpenFingersServiceRelease : BOOL;
	sealFlattenersServiceRaise : BOOL;
	sealFlattenersServiceLower : BOOL;
	sealFlattenersServiceJogIn : BOOL;
	sealFlattenersServiceJogOut : BOOL;
	sealFlattenersManualPositionSetting : REAL;
	sealFlattenersMoveToManualPos : BOOL;
	passthroughManualPositionSetting : REAL;
	passthroughMoveToManualPos : BOOL;
	factoryTestMode : BOOL;
	vacuumServiceOn : BOOL;
	vacuumServiceOff : BOOL;
	printHeadServiceRaise : BOOL;
	printHeadServiceLower : BOOL;
	externalExitConveyorStart : BOOL;
	externalExitConveyorStop : BOOL;
	externalExitConveyorJog : BOOL;
	externalExitConveyorStartDwell : BOOL;
	triggerBarcodeReaderService : BOOL;
	
	(*Factoy Config*)
	bofSelection : BagOpenFingersSelection := BagOpenFingersSelection.PneumaticWithBagOpenSensors;
	sealFlattenersSelection : SealFlattenerSelection := SealFlattenerSelection.MotorizedSealFlatteners;
	printerSelection : LabelPrinterSelection := LabelPrinterSelection.ZebraPrinter203DPI;
	integratedExitConveyorSelection : IntegratedConveyorSelection := IntegratedConveyorSelection.RearExit;
	externalExitConveyorSelection : ExteralConveyorSelection := ExteralConveyorSelection.NotInstalled;
	packageEjectSelection : PackageEjectionSelection := PackageEjectionSelection.RearRetractingLoadPlate;
	independentBagDeflatorSelection : BagDeflatorSelection := BagDeflatorSelection.NotInstalled;
	cycleStartButtonSelection : PalmButtonSelection := PalmButtonSelection.DualPalmButton;
	barcodeVerifierSelection : BCVSelection := BCVSelection.NotInstalled;
	baggerModelSelection : ModelSelection;
	auxIOConfig : AuxIOConfiguration;
	fillerFactorySelection : FillerSelection;
	funnelFactorySelection : FunnelSelection;
	murrIOConfigVersion : CONFIG_VERSIONS := CONFIG_VERSIONS.V_1_3;
	printerConfigVersion : CONFIG_VERSIONS := CONFIG_VERSIONS.V_1_2;
	frontFilmFeedMotorConfigVersion : CONFIG_VERSIONS := CONFIG_VERSIONS.V_1_0;
	rearUnwindMotorConfigVersion : CONFIG_VERSIONS := CONFIG_VERSIONS.V_1_1;
	sealFlattenerMotorConfigVersion : CONFIG_VERSIONS := CONFIG_VERSIONS.V_1_0;
	
	(*Warnings*)
	printerRibbonLow : Warning;
	printerNotReady : Warning;
	waitingForPrinter : Warning;
	sealBarNotAtTemperature : Warning;
	recoveryModeActive : Warning;
	jobLoadRequired : Warning;
	baggerNotReady : Warning;
	demoModeIsActive : Warning;
	factoryTestModeActive : Warning;
	machineNotTested : Warning;
	packageEjectGuardRemoved : Warning;
	bagLevelLow : Warning;
	fillerModeCycleStartOnly : Warning;
	baggerInhibited : Warning;
	infeedConveyorOutOfParts : Warning;
	mayCycleUnexpectedly : Warning;
	(*Misc*)
	pressureBarState : STRING;
    
    (*Counters*)
    baggerCycles : FB_CycleCounter;
	bagOpenFingerCycles : FB_CycleCounter;
	bagsMade : FB_CycleCounter;
	sealBarCycles : FB_CycleCounter;
	pressureBarCycles : FB_CycleCounter;
	passthroughChanges : FB_CycleCounter;
	loadPlateCycles : FB_CycleCounter;
	printerCycles : FB_CycleCounter;
	motorizedSealFlattenerCycles : FB_CycleCounter;
	bagOpenRetryTotal : FB_CycleCounter;
	bagsRejectedTotal : FB_CycleCounter;
	resettableBagsMade : FB_CycleCounter;
	
	(*Predictive Maint.*)
	airFilterClean : FB_PredictiveMaint := (target := 30000, count := 0, name := 'Clean Air Filter');
	driveRollerClean : FB_PredictiveMaint := (target := 20000, count := 0, name := 'Clean Drive Rollers', units := 'Inches of Bag');
	printHeadClean : FB_PredictiveMaint := (target := 10000, count := 0, name := 'Clean Print Head', units := 'Printer Cycles');
	pressureBarGuideShaftGuides : FB_PredictiveMaint := (target := 0, count := 127888, name := 'Replace Guide Shafts');
	
	pressureBarLeak : FB_CylinderLeak := (maximumStrokeTime := 5.0, name := 'Pressure Bar Stroke', units := 'Seconds');
	loadPlateLeak : FB_CylinderLeak := (maximumStrokeTime := 2.0, name := 'Load Plate Stroke', units := 'Seconds');
	
	msfHorizontalMotorTemp : FB_DriveTemp := (maxTemp := 60.0, name := 'MSF Motor Temp.', units := 'deg C');
	bagDeliveryMotorTemp : FB_DriveTemp := (maxTemp := 60.0, name := 'Bag Delivery Motor Temp.', units := 'deg C');
	passthroughMotorTemp : FB_DriveTemp := (maxTemp := 60.0, name := 'Passthrough Motor Temp.', units := 'deg C');
	
	(*Info*)
	faultActive : BOOL;

END_VAR

VAR_GLOBAL CONSTANT
	murrIOConfigVersionMax : CONFIG_VERSIONS := CONFIG_VERSIONS.V_1_3;
	printerConfigVersionMax : CONFIG_VERSIONS := CONFIG_VERSIONS.V_1_2;
	frontFilmFeedMotorConfigVersionMax : CONFIG_VERSIONS := CONFIG_VERSIONS.V_1_0;
	rearUnwindMotorConfigVersionMax : CONFIG_VERSIONS := CONFIG_VERSIONS.V_1_1;
	sealFlattenerMotorConfigVersionMax : CONFIG_VERSIONS := CONFIG_VERSIONS.V_1_0;
END_VAR

// Globals
{attribute 'qualified_only'}
VAR_GLOBAL
    firstScan : BOOL; //First Scan Bit
    pressureBarServoCommsType : MODBUS_COMM_TYPE;  //Comm path to Pressure Bar Servo - 0 = TCP, 1 = RTU
    STEPS_PER_INCH : INT;  //Steps Per Inch for Pressure Bar Servos
    enableDryCycle : BOOL;          // Enable dry cycle
	SystemLog : FB_InternalLogger;
	jawMovingIn : BOOL;
	passthroughChangedFromJog : BOOL;
	machinePowerOK : BOOL;
END_VAR

VAR_GLOBAL CONSTANT
    STEPS_PER_INCH_SEAL_FLATTENER_HORIZONTAL_AXIS_MOTOR  : INT := 2500;
    STEPS_PER_INCH_SEAL_FLATTENER_VERTICAL_AXIS_MOTOR : INT := 2890;        //Steps per inch for NEMA 17 seal flattener finger motor
    STEPS_PER_INCH_BIG_MOTOR : INT := 21872;        //Steps per inch for NEMA 17 motor
    STEPS_PER_INCH_SMALL_MOTOR : INT := 19600;        //Steps per inch for NEMA 11 motor
    STEPS_PER_INCH_SHOW_MOTOR : INT := 18900;        //Steps per inch for NEMA 11 motor
    STEPS_PER_INCH_PRINTER : INT := 4498;            //Steps per inch for printer step servo
    STEPS_PER_INCH_20_DEGREE_BAG_DELIVERY : INT := 5093; // Steps per inch for 20 degree bag delivery motors
	STEPS_PER_INCH_PRO24_BAG_DELIVERY : INT := 4428; // Steps per inch for 20 degree bag delivery motors
	STEPS_PER_INCH_ADJUSTABLE_PASSTHROUGH : INT := 3030;  // Steps per inch for the Adjustable Passthrough motor
	STEPS_PER_INCH_TFBelt : INT := 3030;  // Steps per inch for the Adjustable Passthrough motor
	STEPS_PER_INCH_TFLS : INT := 10000;  // Steps per inch for the Adjustable Passthrough motor
    VELOCITY_IPS_MULTIPLIER_20_DEGREE_BAG_DELIVERY: REAL := 53;
    PASSTHROUGH_ZERO_OFFSET : REAL := 2;            //Zero offset for passthough (minimum passthough)
    MAX_BAG_WIDTH : REAL := 18;                //Passthrough setting
	AMP_MOTOR_RPI : INT := 10;
	MAX_LOGGED_ITEMS : UINT := 500;	// Max items to be logged
END_VAR

VAR_GLOBAL
    headCycleCount : DINT;                 // Head Cycle Counts
	headCycleCount2 : DINT;                 // Head Cycle Counts
    bagGrabberCycleCount : DINT;         // Bag Grabber Cycle Counts
    solenoidCycleCount1 : DINT;         // Solenoid Cycle Cycle Counts (first solenoid)
    motorizedSealFlattenersCount : DINT;         // MSF Cycle Counts
    bagOpenFingersCount : DINT;        // Bag Open Finger Cycles
    sealFlattenerFingersCount : DINT;  // Seal Flattener Fingers Cycle Count
    electricPressureBarCount : DINT;    // Electric Pressure bar Cycle count
    sealBarCount : DINT;                 // Seal bar Cycle count
    bagDeliveryCycleCount : DINT;        // Bag Delivery Cycle Count
    printerCycleCounts : DINT;            // Printer Cycle Counts
    bagsMadeCount : DINT;                // Bags Made
    passthroughChangeCount : DINT;        // Passthrough Changes
	passthroughChangeDistance : UDINT;	// Passthrough Distance Changes in .1 Inches
	solenoidCycleCount2 : DINT;     	// Solenoid Cycle Cycle Counts (Strech SX)	
	solenoidFailureCount2 : UDINT;		// Solenoid Failure Count (Strech SX)
	pickAndPlaceCycleCount : UDINT;		// Pick and place cycle count
	passthroughChangeCount2 : DINT;        // Passthrough Changes
	passthroughChangeDistance2 : UDINT;	// Passthrough Distance Changes in .1 Inches
	bagFailedToGrabBothFingersCount : UDINT; // Both Fingers failed to grab bag
	bagFailedToGrabRightFingerCount : UDINT; // Right Bag Open Finger Failed to Grab Bag
	bagFailedToGrabLeftFingerCount : UDINT; // Left Bag Open Finger Failed to Grab Bag
	successfulBagOpenCount : UDINT;			// Successful Bag Open Count
	rejectedBagCount : UDINT;				// Rejected bag count 
    dryCycleCount  :UDINT;                   // Dry cycle count
	lastPrinterDelta : TIME := T#100MS;
	factoryTestComplete : BOOL;		// 1000 bags test done
END_VAR

// Pro18_1174/Application/Programs/PRG_MainProgram
PROGRAM PRG_MainProgram
VAR
    incrementSolenoidCounter1 : R_TRIG();
    incrementSolenoidCounter2 : R_TRIG();
    incrementSolenoidFailedCounter2 : R_TRIG();
    GripperCycleCount : DINT; //Gripper Cycle Counter
    runPrinterPB : BOOL;
    cycleTimeMax : TIME;
    cycleTimeMaxDINT : DINT;
    ctfb : OSCAT_BASIC.CYCLE_TIME();
    profileThis :BOOL;
    solenoidState1 : SOLENOID_TEST_STATES;
    solenoidState2 : SOLENOID_TEST_STATES;
    getTimeTilPMMI : TimeLeftFB();
	displayPassthroughChangeDistance : REAL;
	displayPassthroughChangeDistance2 : REAL;
	checkSolenoid2ExtendTimer : TON := (PT := T#100MS);
	checkedSolenoid2Status : BOOL;
	firstScanDone : BOOL;
	printDeltaTimer : TON := (PT := T#5S);
	lastPrinterDelta : TIME;
	endPrintOSF : Standard.R_TRIG;
	stringToLog : STRING;
	testWrite : BOOL;
	hmiLight : FB_HMILight;
	versionInfo : VERSION;
	recipieManager : Recipe_Management.RecipeManCommands;
	recipeName : STRING;
	recResult : DWORD;
	testRead : BOOL;
	testCreate : BOOL;
	saveParametersTimer : Standard.TON := (PT := T#10M);
	EIPReconfig : FB_EIPCommsConfigure();
END_VAR

//    Program: Main (PLC_PRG)
//    Description: This program serves as a base for the MOAB Prototype
//    Created by: Ben Hess
//    Created Date: January 16th, 2018

printDeltaTimer(IN := oPrinterStartPrint);
saveParametersTimer(IN := NOT saveParametersTimer.Q);
IF saveParametersTimer.Q THEN
	recResult := recipieManager.GetRecipeNames('Recipes', ADR(recipeName),1,0);
	recResult := recipieManager.ReadAndSaveRecipe(RecipeDefinitionName := 'Recipes', RecipeName := recipeName);
	saveParametersTimer.IN := FALSE;
END_IF
EIPReconfig(rootEIPNode := CIFX_EIP);
IF testCreate THEN
// 	recResult := recipieManager.CreateRecipe(RecipeDefinitionName := 'Recipes', RecipeName := 'Automatic');
// 	recResult := recipieManager.ReadAndSaveRecipe(RecipeDefinitionName := 'Recipes', RecipeName := recipeName);
 	testCreate := FALSE;
	SaveValues();
END_IF

IF testRead THEN
// 	recResult := recipieManager.GetRecipeNames('Recipes', ADR(recipeName),1,0);
// 	recResult := recipieManager.LoadAndWriteRecipe(RecipeDefinitionName := 'Recipes', RecipeName := recipeName);
 	testRead := FALSE;
	RecallValues();
END_IF

// 
// CSVWriter(
// 	xFilePath:= , 
// 	xText_Write:= , 
// 	xAppend_OverWrite:= TRUE, 
// 	xAppend_Pos:= , 
// 	xWrite:= , 
// 	xRead:= , 
// 	xLine_No_To_Read:= , 
// 	xText_Read=> , 
// 	xDone=> );
// IF CSVWriter.xDone THEN
// 	CSVWriter.xWrite := FALSE;
// END_IF

ctfb(ct_max => cycleTimeMax);
cycleTimeMaxDINT := TIME_TO_DINT(cycleTimeMax);
profileThis := TIME_TO_DINT(ctfb.ct_last) >= 25;
// Run other programs
//PRG_PneumaticHead();
PRG_Bagger();
Faults();
versionInfo := GetVersion();
HMIData.version := Standard.CONCAT(TO_STRING(versionInfo.uiMajor),'.');
	BPLog.AppendToString(ADR(HMIData.version), CONCAT(TO_STRING(versionInfo.uiMinor),'.'));
	BPLog.AppendToString(ADR(HMIData.version), CONCAT(TO_STRING(versionInfo.uiServicePack),'.'));
	BPLog.AppendToString(ADR(HMIData.version), TO_STRING(versionInfo.uiPatch));
	BPLog.AppendToString(ADR(HMIData.version), TO_STRING(GetTextProperty("VersionPostfix")));
IF NOT firstScanDone THEN
	GlobalObjects.CollectionOfLoggable.RegisterAll(internalLogger := Globals.SystemLog);
	GlobalObjects.CollectionOfInitialzable.InitializeAll();
	firstScanDone := TRUE;
	// After first scan turn off flag set by StartDone system event
	Globals.firstScan := FALSE;	
END_IF

// Start executing objects that implement IExecuteAutomatically 
IF firstScanDone THEN
	GlobalObjects.CollectionOfExecutable.ExecuteAll();
	Globals.SystemLog();
END_IF




IF HMIData.ackAllFaults THEN
	GlobalObjects.CollectionOfActiveFaults.AckAll();
	HMIData.ackAllFaults := FALSE;
END_IF

getTimeTilPMMI(targetDate := DT#2018-10-14-8:0:0);


//First scan flag is set by task handler and reset in main routine here
IF Globals.firstScan THEN
    Globals.firstScan := FALSE;
END_IF

displayPassthroughChangeDistance := (UDINT_TO_REAL(Globals.passthroughChangeDistance) / 10);
displayPassthroughChangeDistance2 := (UDINT_TO_REAL(Globals.passthroughChangeDistance2) / 10.0);

END_PROGRAM

// Pro18_1174/Application/SaveValues
FUNCTION SaveValues : DWORD
VAR
	recipieManager : Recipe_Management.RecipeManCommands;
	recipeName : STRING;
	recResult : DWORD;
END_VAR

recResult := recipieManager.CreateRecipe(RecipeDefinitionName := 'Recipes', RecipeName := 'Automatic');
recResult := recipieManager.GetRecipeNames('Recipes', ADR(recipeName),1,0);
recResult := recipieManager.ReadAndSaveRecipe(RecipeDefinitionName := 'Recipes', RecipeName := recipeName);

END_FUNCTION

// ElectricMachine/Application/SaveValues
FUNCTION SaveValues : DWORD
VAR
	recipieManager : Recipe_Management.RecipeManCommands;
	recipeName : STRING;
	recResult : DWORD;
END_VAR

//IF HMIData.bagsMade.count <> 0 THEN
	recResult := recipieManager.CreateRecipe(RecipeDefinitionName := 'Recipes', RecipeName := 'Automatic');
	recResult := recipieManager.GetRecipeNames('Recipes', ADR(recipeName),1,0);
	recResult := recipieManager.ReadAndSaveRecipe(RecipeDefinitionName := 'Recipes', RecipeName := recipeName);
//END_IF

END_FUNCTION

// Pro18_1174/Application/RecallValues
FUNCTION RecallValues : DWORD
VAR
	recipieManager : Recipe_Management.RecipeManCommands;
	recipeName : STRING;
	recResult : DWORD;
END_VAR

recResult := recipieManager.GetRecipeNames('Recipes', ADR(recipeName),1,0);
recResult := recipieManager.LoadAndWriteRecipe(RecipeDefinitionName := 'Recipes', RecipeName := recipeName);

END_FUNCTION

// ElectricMachine/Application/RecallValues
FUNCTION RecallValues : DWORD
VAR
	recipieManager : Recipe_Management.RecipeManCommands;
	recipeName : STRING;
	recResult : UDINT;
END_VAR

recResult := recipieManager.CreateRecipe(RecipeDefinitionName := 'Recipes', RecipeName := 'Automatic');
recResult := recipieManager.GetRecipeNames('Recipes', ADR(recipeName),1,0);
recResult := recipieManager.LoadAndWriteRecipe(RecipeDefinitionName := 'Recipes', RecipeName := 'Automatic');

END_FUNCTION

// ElectricMachine/Application/Programs/PRG_Bagger
PROGRAM PRG_Bagger
VAR_INPUT

END_VAR
VAR_OUTPUT
    
END_VAR
VAR
    moabHead : FB_MOABHead_Electric;
    //angledHead : FB_20degHead();
    //pneuHead : FB_PneumaticHead();
    testEIPMotor : FB_AppliedMotionStepServoEIPBase();
    faultHandler : FB_FaultHandler();
	hmiInitiate : BOOL;
	msfMotorFaults : ARRAY[0..100] OF MotorCommFault;
	numberOfMSFFaults : UINT;
	msfCommFaultONS : R_TRIG();
	msfFaultListFull : BOOL;
	festoFaults : ARRAY[0..100] OF MotorCommFault;
	numberOfFestoFaults : UINT;
	festoCommFaultONS : R_TRIG();
	festoFaultListFull : BOOL;
	currentDateAndTime : GetTime();
	resetCommFaults : BOOL;
	i : INT;
	reverseFault : FB_HMIFault := (refFault := PRG_Bagger.moabHead.bagDelivery.reverseFault);
	faultActiveONS : FB_ONS;
	

END_VAR

//    Program: PRG_Bagger 
//    Description: This program glues together the whole machine and all of its components.
//    
//    Created by: Ben Hess
//    Created Date: Tuesday, April 17, 2018

moabHead();
//pneuHead();
faultHandler();
hmiInitiate := HMIData.initiateCycle;
currentDateAndTime();
//msfCommFaultONS(CLK := MSFMotor.eState <> IoDrvEthernetIP.AdapterState.RUNNING);
HMIData.bagEdgePhotoeyeCovered := NOT iBagNotPresent;
oSoftStart := TRUE;

HMIData.airFilterClean();
HMIData.pressureBarGuideShaftGuides();
HMIData.driveRollerClean();
HMIData.printHeadClean();
//HMIData.pressureBarLeak(iExtended := iPressureBarExtended, iRetracted := iPressureBarRetracted, maximumStrokeTime := (TO_REAL(HMIData.passthroughSetting / 26.6)) + 0.3);
HMIData.loadPlateLeak(iExtended := iLoadPlateExtended, iRetracted := iLoadPlateRetracted, maximumStrokeTime := 0.4);
//HMIData.msfHorizontalMotorTemp(iDriveTemp := sealFlattenerHorizontalMotorInputs[4]);
//HMIData.bagDeliveryMotorTemp(iDriveTemp := bagDeliveryMotorInputs[4]);
//HMIData.passthroughMotorTemp(iDriveTemp := jawPasstrhoughMotorInputs[4]);




IF resetCommFaults THEN
	FOR i := 0 TO numberOfMSFFaults BY 1 DO
		msfMotorFaults[i].message := '';
		msfMotorFaults[i].timeOfFault := DT#1970-1-1-1:0:0;
	END_FOR
	numberOfMSFFaults := 0;
	msfFaultListFull := FALSE;
	resetCommFaults := FALSE;
END_IF


//HMIData.version := SVN_VERSION_INFO.VERSION;

HMIData.faultActive := GlobalObjects.CollectionOfActiveFaults.faultActive;
faultActiveONS(CLK := GlobalObjects.CollectionOfActiveFaults.faultActive);
IF faultActiveONS.OSR THEN
	moabHead.hmiLight.TurnOff();
END_IF

END_PROGRAM

// Pro18_1174/Application/Programs/PRG_Bagger
PROGRAM PRG_Bagger
VAR_INPUT

END_VAR
VAR_OUTPUT
    
END_VAR
VAR
    moabHead : FB_MOABHead;
    //angledHead : FB_20degHead();
    //pneuHead : FB_PneumaticHead();
    testEIPMotor : FB_AppliedMotionStepServoEIPBase();
    faultHandler : FB_FaultHandler();
	hmiInitiate : BOOL;
	msfMotorFaults : ARRAY[0..100] OF MotorCommFault;
	numberOfMSFFaults : UINT;
	msfCommFaultONS : R_TRIG();
	msfFaultListFull : BOOL;
	festoFaults : ARRAY[0..100] OF MotorCommFault;
	numberOfFestoFaults : UINT;
	festoCommFaultONS : R_TRIG();
	festoFaultListFull : BOOL;
	currentDateAndTime : GetTime();
	resetCommFaults : BOOL;
	i : INT;
	reverseFault : FB_HMIFault := (refFault := PRG_Bagger.moabHead.bagDelivery.reverseFault);
	faultActiveONS : FB_ONS;
END_VAR

//    Program: PRG_Bagger 
//    Description: This program glues together the whole machine and all of its components.
//    
//    Created by: Ben Hess
//    Created Date: Tuesday, April 17, 2018

moabHead();
//pneuHead();
faultHandler();
hmiInitiate := HMIData.initiateCycle;
currentDateAndTime();
//msfCommFaultONS(CLK := MSFMotor.xDiagnosticAvailable);
HMIData.bagEdgePhotoeyeCovered := NOT iBagNotPresent;
oSoftStart := TRUE;

HMIData.airFilterClean();
HMIData.pressureBarGuideShaftGuides();
HMIData.driveRollerClean();
HMIData.printHeadClean();
HMIData.pressureBarLeak(iExtended := iPressureBarExtended, iRetracted := iPressureBarRetracted, maximumStrokeTime := (TO_REAL(HMIData.passthroughSetting / 26.6)) + 0.3);
HMIData.loadPlateLeak(iExtended := iLoadPlateExtended, iRetracted := iLoadPlateRetracted, maximumStrokeTime := 0.4);
//HMIData.msfHorizontalMotorTemp(iDriveTemp := sealFlattenerHorizontalMotorInputs[4]);
//HMIData.bagDeliveryMotorTemp(iDriveTemp := bagDeliveryMotorInputs[4]);
//HMIData.passthroughMotorTemp(iDriveTemp := jawPasstrhoughMotorInputs[4]);




IF resetCommFaults THEN
	FOR i := 0 TO numberOfMSFFaults BY 1 DO
		msfMotorFaults[i].message := '';
		msfMotorFaults[i].timeOfFault := DT#1970-1-1-1:0:0;
	END_FOR
	numberOfMSFFaults := 0;
	msfFaultListFull := FALSE;
	resetCommFaults := FALSE;
END_IF

//HMIData.version := SVN_VERSION_INFO.VERSION;

HMIData.faultActive := GlobalObjects.CollectionOfActiveFaults.faultActive;
faultActiveONS(CLK := GlobalObjects.CollectionOfActiveFaults.faultActive);
IF faultActiveONS.OSR THEN
	moabHead.hmiLight.TurnOff();
END_IF

END_PROGRAM

// FBs/FunctionalAreas/FB_MOABHead
FUNCTION_BLOCK FB_MOABHead EXTENDS BaseComponentFB
VAR_INPUT
    motorizedSealFlattenersMode : DEVICE_MODES := DEVICE_MODES.Auto;
    electricPressureBarMode : DEVICE_MODES := DEVICE_MODES.Auto;
	vacuumPickerMode : DEVICE_MODES;
    startCycle : BOOL;
    bagDeliveryMode : DEVICE_MODES;        // Mode of bag delivery system
    printerMode : DEVICE_MODES;        // Mode of printer
	passthroughMode : DEVICE_MODES;
    batchSetting : DINT;            // Batch setpoint
    batchCount : DINT;                // Actual batch cycles
    enableBatch : BOOL;                // Enable Batch Mode
    enableBatchONS : F_TRIG;
	passthroughSetting : REAL;
    passthroughSettingLast : REAL;
	bagDropDelay : UINT := 1000;
END_VAR
VAR_OUTPUT
    readyToRun : BOOL;
    state : HEAD_STATES;
    sealAndSeparateSubState : SEAL_SEPARATE_STATES;
    releaseAndFeedSubState : RELEASE_FEED_STATES;
    openBagSubState : BAG_OPEN_ASSIST_STATES;
	finishCycleSubState : FINISH_CYCLE_STATES;
END_VAR
VAR
    motorizedSealFlatteners : MotorizedSealFlattenersFB_BagFeed();
	msfVerticalAxis : FB_ThreePositionCylinder();
    pressureBar : PneumaticPressureBarFB_1();
	sealBarTempSensor : FB_IFMTempSensor();
	sealBarHeater : FB_TempController();
    startCycleONS : R_TRIG;
	enableBagOpen : BOOL;
	enableLoadPlate : BOOL;
	enableHeater : BOOL;
	enableIBDDeflate : BOOL;
	enableIBDEject : BOOL;
	enableLabelSideUp : BOOL := TRUE;
	factoryTestModeKeepCycling : BOOL;
    bagDelivery : BagDeliveryFB();
    //zebraPrinter : PrinterFB;            //Printer Test Rig
	zebraPrinter : PrinterFB_Mode2;
	sealTimer : Standard.TON() := (PT := T#350MS);
	bagOpenFingerDelay : Standard.TON := (PT := T#100MS);
	bagDropTimer : Standard.TON;
	HPA : MonostableMultivibratorFB();
    rearLoadPlateRetract : MonostableMultivibratorFB() := (Dwellsetting := 1500);
	forwardLoadPlateRetract : MonostableMultivibratorFB() := (Dwellsetting := 1500);
	loadShelfExtend : MonostableMultivibratorFB() := (Dwellsetting := 1500);
	exitConveyorRun : DelayDwellFB() := (Dwellsetting := 6000);
	externalExitConveyorRun : DelayDwellFB() := (Dwellsetting := 6000);
	IBDCylinders : FB_ThreePositionCylinder();
	IBDExtendONS : FB_ONS();
	IBDRetractONS : FB_ONS();
	IBDRetractToDeflate : MonostableMultivibratorFB();
	IBDRetractToEject : MonostableMultivibratorFB();
	bagOpenFingers : BagOpenFingersWithSensorsFB();
	bagOpenCheckDelay : Standard.TON := (PT:= T#400MS); // Delay to check if bag open
	bagOpenRetrySetting : UINT;		// Number of times to retry opening bag
	bagOpenRetryCount : UINT;		// Count of current retry attempts
	bagOpenFeedNewBagSetting : UINT; // Number of new bags to try
	bagOpenFeedNewBagCount : UINT;	// Count of new bags tried in recovery
	bagOpened : BOOL;				// Bag was Opened flag
	recoveryModeActive : BOOL; 		// Recovery Mode Active
	startCycleReqFromPalmButtons : BOOL;
	startCycleReqFromPalmButtonsONS : FB_ONS();
	pressureBarEndStopMotor : FB_AppliedMotionStepServoEIPPassthrough();
	passthrough : AdjustablePassthroughFB();
	homeJawPB : BOOL;
    setPassthroughPB : BOOL;
	vacuumHoldTimer : Standard.TON() := (PT := T#250MS);
	cycleTimer : TON() := (PT := T#1000S);
	cycleTime : REAL;
	bagFailedToOpen : FB_Fault(name := 'Bag Failed to Open');
	openedBagWasRemoved : FB_Fault(name := 'Opened Bag was Removed');
	safePowerFailure : FB_Fault(name := 'E-Stop/Safety Power Failure');
	palmButtonConfigError : FB_Fault(name := 'Palm Button Configuration Error');
	packageEjectGuardRemoved : FB_Fault(name := 'Package Eject Guard Removed');
	barcodeVerificationFailed : FB_Fault(name := 'Barcode Verification Failed');
	barcodeVerifierCommFail : FB_Fault(name := 'Barcode Verifier Communication Failure');
	infeedConveyorIOCommFail : FB_Fault(name := 'Infeed Conveyor IO Communication Failure');
	infeedConveyorVFDFaulted : FB_Fault(name := 'Infeed Conveyor VFD Failure');
	iPowerOffButtonONS : FB_ONS();
	loadPlateFaultTimer : FB_CylinderFaults();
	loadPlateFaults : LoadPlateFaultsType;
	forwardLoadPlateFaultTimer : FB_CylinderFaults();
	forwardLoadPlateFaults : LoadPlateFaultsType;
	rearLoadPlateFaultTimer : FB_CylinderFaults();
	rearLoadPlateFaults : LoadPlateFaultsType;
	loadShelfFaultTimer : FB_CylinderFaults();
	loadShelfFaults : LoadPlateFaultsType;
	LPA : DelayDwellFB();
	hpaServiceOnONS : FB_ONS;
	exitConveyorJogONS : FB_ONS;
	externalExitConveyorJogONS : FB_ONS;
	hmiLight  : FB_HMILight;
	faultONS : FB_ONS;
	powerSettlingTimer : Standard.TON := (PT := T#6S);
	pressureBarCloseDelay : Standard.TON;
	filler : FillerFB();
	configOutput1Pulse : MonostableMultivibratorFB();
	configOutput2Pulse : MonostableMultivibratorFB();
	fillerModeCycleStartOnlyPulse : MonostableMultivibratorFB();
	murrIOBusNode : MurrIOFB();
	funnel : FunnelFB();
	barcodeVerifier : BarcodeReaderFB();
	keyenceBCV : KeyenceNL20FB();
	rearMotorCommsReturned : Standard.F_TRIG();
	ezfeed : EZFeedFB();
END_VAR

//    Function Block: FB_MOABHead
//    Description: This is the supervisory module for the MOAB head.
//    There is one supervisory state machine for the head and 3 sub-state machines Sealing/Separating, Release/Feed, and Opening Bag
//    Created by: Ben Hess
//    Created Date: Tuesday, April 17, 2018

{region "Setup"}
// Run BaseComponentFB
SUPER^();

// When power is returned, give machine ~5 seconds
powerSettlingTimer(IN := iEStopOK);
Globals.machinePowerOK := powerSettlingTimer.Q;
safePowerFailure.faultTrigger := NOT iEStopOK AND murrIOBusNode.ok;

// Bags Low warning
HMIData.bagLevelLow.active := iBagsLow;

// Ethernet/IP barcode verifier from Keyence
keyenceBCV(
	enable:= , 
	ptrEIPInputs:= ADR(keyenceBCVInputs), 
	ptrEIPOutputs:= ADR(keyenceBCVOutputs), 
	triggerInput:= , 
	//commFail=> ,
	lastReadData => HMIData.barcodeLastReadString);	 
// Barcode Verifier interface to printer
barcodeVerifier(enable := (HMIData.barcodeVerifierSelection <> BCVSelection.NotInstalled AND HMIData.barcodeVerifierInUse),
		 		readGoodInput := keyenceBCV.goodRead,
				distanceToScan := HMIData.barcodeScanDistance,
				feedSpeed := TO_REAL(HMIData.printSpeed),
				positionOffset := HMIData.barcodeStartPosition,
				badReadFaultCountSetting := HMIData.barcodeBadReadFaultSetting,
				currentBadReadCount => HMIData.barcodeBadReadCount,
				currentGoodReadCount => HMIData.barcodeGoodReadCount,
				triggerScannerOutput => keyenceBCV.triggerInput);
// Enable comms to Keyence N-L20 if selected in factory config
IF HMIData.barcodeVerifierSelection = BCVSelection.LaserScanner THEN
	Keyence_BCV.Enable := TRUE; 

	IF Keyence_BCV.udiState <> 4 THEN 
		barcodeVerifierCommFail.Trigger();
	END_IF

ELSE
	Keyence_BCV.Enable := FALSE;
END_IF


// Option setup and factory config  
	 
IF HMIData.resetAverageCycleTime THEN
	HMIData.averageCycleTime := 0;
	HMIData.resetAverageCycleTime := FALSE;
END_IF
HMIData.lastCycleTime := cycleTime;

HMIData.printerNotReady.active := NOT printerReady AND zebraPrinter.enable;
HMIData.waitingForPrinter.active := zebraPrinter.state = PRINTER_STATES.WaitingForData AND releaseAndFeedSubState = RELEASE_FEED_STATES.WaitForPrinter;
//HMIData.printerRibbonLow.active := printerRibbonLow;
	 
batchSetting := HMIData.batchSetting;
HMIData.batchCount := batchCount;

bagOpenRetrySetting := HMIData.bagOpenRetrySetting;
HMIData.bagOpenRetryCount := bagOpenRetryCount;
	 
// Run bus node		  
murrIOBusNode(
	enable:= , 
	headNodeEnabled:= TRUE, 
	guardNodeEnabled:= (HMIData.cycleStartButtonSelection <> PalmButtonSelection.NotInstalled) OR (HMIData.funnelFactorySelection <> FunnelSelection.NotInstalled), 
	printerNodeEnabled:= (HMIData.printerSelection <> LabelPrinterSelection.NotInstalled), 
	dischargeNodeEnabled:= TRUE, 
	auxIONodeEnabled:= , 
	configVersion:= HMIData.murrIOConfigVersion, 
	ptrMachineOptionsManagementOutputs:= ADR(oMOMConfig), 
	ptrSystemStatusInputs:= ADR(iMurrSystemState));

// Setup of Motorized seal flattener motor and function block
msfVerticalAxis(extendOutput => oSealFlatDown, retractOutput => oSealFlatUp);
msfVerticalAxis.Execute();
motorizedSealFlatteners(sealFlattenersVerticalAxis := msfVerticalAxis,
						jogIn := HMIData.sealFlattenersServiceJogIn,
						jogOut := HMIData.sealFlattenersServiceJogOut,
						raiseService := HMIData.sealFlattenersServiceRaise,
						lowerService := HMIData.sealFlattenersServiceLower,
						moveToManualSetpoint := HMIData.sealFlattenersMoveToManualPos,
						manualPosSetpoint := HMIData.sealFlattenersManualPositionSetting,
						sealFlattenerMotorCommFailInput := MSFMotor.udiState <> 4);
motorizedSealFlatteners.Mode := motorizedSealFlattenersMode;

// Setup of MOAB Machine Pressure bar ("#2") on actual machine, not test rig
pressureBar(iPressureBarExtended := iPressureBarExtended, 
			iPressureBarRetracted := iPressureBarRetracted, 
			iPressureBarNotObstructed := iPressureBarNotObstructed, 
			oExtendCylinder => oPBar1Extend, oRetractCylinder => oPBar1Retract,
			cumulativeHeadCycleCount := Globals.headCycleCount2);
pressureBar.Mode := electricPressureBarMode;
//Adding extra pressure bar valve for test
opBar2Extend := oPBar1Extend;
opbar2Retract := oPBar1Retract;


// Run bag delivery 
bagDelivery(jogForwardPB := HMIData.jogBagForward,
			jogReversePB := HMIData.jogBagReverse,
			bagFeedMasterMotorCommFailInput := Bag_Delivery_EIP_Motor.udiState <> 4,
			bagFeedRearMotorCommFailInput := Bag_Delivery_Rear_Motor.udiState <> 4,
			stepsPerInchSetting := Globals.STEPS_PER_INCH_20_DEGREE_BAG_DELIVERY);
bagDelivery.Mode := bagDeliveryMode;

// Run Zebra Printer
zebraPrinter(ribbonEncoderPulse := iPrinterRibbonEncoder, oLowerPrintHead => oPrintHeadDown);
zebraPrinter.Mode := printerMode;
zebraPrinter.enable := (HMIData.printerSelection <> LabelPrinterSelection.NotInstalled) AND HMIData.printerInUse;
IF HMIData.activateDemoMode THEN
	HMIData.demoModeIsActive.active := TRUE;
	zebraPrinter.autoSendLabel := TRUE;
ELSE
	HMIData.demoModeIsActive.active := FALSE;
	zebraPrinter.autoSendLabel := FALSE;
END_IF

	 
// Run funnel
funnel(
	enable:= HMIData.funnelFactorySelection <> FunnelSelection.NotInstalled AND HMIData.funnelInUse, 
	sensorsInstalled:= HMIData.funnelFactorySelection = FunnelSelection.FunnelWithSensors, 
	openSensor:= iFunnelOpened, 
	closedSensor:= iFunnelClosed, 
	opened=> , 
	closed=> , 
	closeOutput=> oIBDRetract, 
	openOutput=> oIBDExtend, 
	failToOpen=> , 
	failToClose=> );
funnel.OpeningTime := HMIData.funnelOpeningTime;
funnel.ClosingTime := HMIData.funnelClosingTime;
funnel.DelaySetting := HMIData.funnelOpenDelay;
// Setup of pick and place motors


sealBarTempSensor(ptrTemperatureBytes := ADR(iHeaterBarTempInputs));
sealBarTempSensor.Execute();
sealBarHeater(enable := NOT HMIData.faultActive,
				temperatureSensor := sealBarTempSensor,
				temperatureSetpoint := TO_REAL(HMIData.sealBarTemperatureSetting),
				heaterPulse => 	oHeaterPulse);	  
HMIData.sealBarTemperature := TO_UDINT(sealBarHeater.currentTemp);
{region "timers"}
// Timers
sealTimer();
bagOpenFingerDelay();
vacuumHoldTimer(PT := TO_TIME(HMIData.vacuumDwell * 1000));
bagOpenCheckDelay();
bagDropTimer(PT := TO_TIME((HMIData.loadPlateDelay * 1000) + (HMIData.bagDropTime * 1000)));
{endregion}
		  
// Setup of HPA and load plate.  Use .Trigger() to run.
HPA.DwellSetting := TO_UINT(HMIData.hpaDwell * 1000);
HPA(Q => oHPAOn);
hpaServiceOnONS(CLK := HMIData.hpaserviceOn);

LPA.DwellSetting := TO_DINT(HMIData.lpaDwell * 1000);
LPA(Q => oLPAOn);
	 
CASE HMIData.independentBagDeflatorSelection OF
	BagDeflatorSelection.NotInstalled:					// Disable IBD
		 													enableIBDDeflate := FALSE;
															enableIBDEject := FALSE;
															IBDRetractToDeflate.DelaySetting := 0;
															IBDRetractToDeflate.DwellSetting := 0;
															IBDRetractToEject.DelaySetting := 0;
															IBDRetractToEject.DwellSetting := 0;
	
	BagDeflatorSelection.IBDStandard:	// Enable IBD
															IBDRetractToDeflate();
															IBDRetractToEject();
															IBDRetractONS(CLK := (IBDRetractToDeflate.Q OR IBDRetractToEject.Q));
															IBDExtendONS(CLK := NOT (IBDRetractToDeflate.Q OR IBDRetractToEject.Q));
																 
															IF HMIData.IBDDeflateDwellTime <> 0 THEN
																enableIBDDeflate := TRUE;
															ELSE
																enableIBDDeflate := FALSE;
															END_IF
															
															IF HMIData.IBDPackageEjectAssistDwellTime <> 0 THEN
																enableIBDEject := TRUE;
															ELSE
																enableIBDEject := FALSE;
															END_IF
	 														IBDCylinders(extendOutput => oIBDExtend, retractOutput => oIBDRetract);
															IF IBDRetractONS.OSR THEN
																IBDCylinders.Retract();
															END_IF
															IF IBDExtendONS.OSR THEN
																IBDCylinders.Extend();
															END_IF
																 
															IBDRetractToDeflate.DelaySetting := 0;
															IBDRetractToDeflate.DwellSetting := TO_UINT(HMIData.IBDDeflateDwellTime * 1000);
															IBDRetractToEject.DelaySetting := TO_UINT(HMIData.IBDPackageEjectAssistDelayTime * 1000);
															IBDRetractToEject.DwellSetting := TO_UINT(HMIData.IBDPackageEjectAssistDwellTime * 1000);
																 
	BagDeflatorSelection.IBDWithHingedPlate:	// Enable IBD with Hinged Plate
															enableIBDDeflate := TRUE;
															IBDCylinders(extendOutput => oIBDExtend, retractOutput => oIBDRetract);	
															oIBDRetract := IBDRetractToDeflate.Q OR IBDRetractToEject.Q;
															oIBDExtend := NOT oIBDRetract;
															IBDRetractToDeflate.DelaySetting := 0;
															IBDRetractToDeflate.DwellSetting := TO_UINT(HMIData.IBDDeflateDwellTime * 1000);
															IBDRetractToEject.DelaySetting := TO_UINT(HMIData.IBDPackageEjectAssistDelayTime * 1000);
															IBDRetractToEject.DwellSetting := TO_UINT(HMIData.IBDPackageEjectAssistDwellTime * 1000);
	
END_CASE

CASE HMIData.bofSelection OF
	BagOpenFingersSelection.NotInstalled:					// Disable Bag Open
		 													enableBagOpen := FALSE;
															
	
	BagOpenFingersSelection.PneumaticWithBagOpenSensors:	// Enable Bag Open
															enableBagOpen := TRUE;
	
END_CASE


CASE HMIData.packageEjectSelection OF
	PackageEjectionSelection.NotInstalled:				// Disable all
														enableLoadPlate := FALSE;
														enableLabelSideUp := FALSE;	
														loadPlateFaultTimer.enable := FALSE;	
														forwardLoadPlateFaultTimer.enable := FALSE;
														rearLoadPlateFaultTimer.enable := FALSE;
														loadShelfFaultTimer.enable := FALSE;
		 
	PackageEjectionSelection.RearRetractingLoadPlate:	// Enable rear retracting load plate
		 												enableLoadPlate := TRUE;
														enableLabelSideUp := FALSE;	
														loadPlateFaultTimer.enable := Globals.machinePowerOK;	
														forwardLoadPlateFaultTimer.enable := FALSE;
														rearLoadPlateFaultTimer.enable := FALSE;
														loadShelfFaultTimer.enable := FALSE;
														rearLoadPlateRetract.DelaySetting := TO_UINT(HMIData.loadPlateDelay * 1000);
														rearLoadPlateRetract.DwellSetting := TO_UINT(HMIData.loadPlateDwell * 1000);
	
	PackageEjectionSelection.LabelSideUp:				// Enable all
		 												enableLoadPlate := TRUE;
														enableLabelSideUp := TRUE;	
														loadPlateFaultTimer.enable := FALSE;
														forwardLoadPlateFaultTimer.enable := Globals.machinePowerOK;
														rearLoadPlateFaultTimer.enable := Globals.machinePowerOK;
														loadShelfFaultTimer.enable := Globals.machinePowerOK;
														rearLoadPlateRetract.DelaySetting := 0;
														rearLoadPlateRetract.DwellSetting := TO_UINT((HMIData.loadPlateDwell + HMIData.loadPlateDelay) * 1000);
END_CASE

CASE HMIData.cycleStartButtonSelection OF
	PalmButtonSelection.NotInstalled:					// Dont' allow input to start bagger cycle
		 												startCycleReqFromPalmButtons := FALSE;
		 
	PalmButtonSelection.SinglePalmButton:				// Start using one side only
		 												startCycleReqFromPalmButtons := iRightPalmButton;
														
														// Trigger fault if left palm button is seen - should be set up for dual!	 
														IF iLeftPalmButton THEN
															palmButtonConfigError.Trigger();		 
														END_IF
		 
	PalmButtonSelection.DualPalmButton:					// Both buttons must be pressed
		 												startCycleReqFromPalmButtons := iRightPalmButton AND iLeftPalmButton;
END_CASE
startCycleReqFromPalmButtonsONS(CLK := startCycleReqFromPalmButtons);	 

CASE HMIData.auxIOConfig.factorySelection OF
	AuxiliaryIOSelection.NotInstalled:					// Turn outputs off
		 												oAuxBaggerOK := FALSE;
														oAuxReadyForFiller := FALSE;
														configOutput1Pulse.ManualOff();	
														configOutput1Pulse.Reset();
														configOutput2Pulse.ManualOff();	
														configOutput2Pulse.Reset();
														murrIOBusNode.auxIONodeEnabled := FALSE;
														HMIData.fillerFactorySelection := FillerSelection.NotInstalled;
		 
	AuxiliaryIOSelection.AuxIOStandard:					// Use aux IO
		 												murrIOBusNode.auxIONodeEnabled := TRUE;
		 												oAuxBaggerOK := NOT HMIData.faultActive;
														oAuxReadyForFiller := filler.waitingForFiller;
															 
 														CASE HMIData.auxIOConfig.cfgInputSelection OF
															AuxInputSelection.NotConfigured:		// 
																									HMIData.baggerInhibited.active := FALSE;
																										 
															AuxInputSelection.BaggerInhibit:		//
																 									HMIData.baggerInhibited.active := iAuxConfigInput;
														END_CASE
 
														CASE HMIData.auxIOConfig.cfgOutput1Selection OF
																 
															AuxOutputSelection.BagMade:				//
																 									IF state = HEAD_STATES.SealedAndSeparatedBag THEN
																										configOutput1Pulse.Trigger();
																									END_IF
																										 
															AuxOutputSelection.CycleComplete:		//
																 									IF state = HEAD_STATES.OpenedBag THEN
																										configOutput1Pulse.Trigger();
																									END_IF
																										 
															AuxOutputSelection.PrinterDataReady:	//
																 									IF printerDataReady THEN
																										configOutput1Pulse.ManualOn();
																									ELSE
																										configOutput1Pulse.ManualOff();
																									END_IF
																										 
															AuxOutputSelection.WaitingForPrinter:	// 
																 									IF releaseAndFeedSubState = RELEASE_FEED_STATES.WaitForPrinter THEN
																										configOutput1Pulse.ManualOn();
																									ELSE
																										configOutput1Pulse.ManualOff();	
																								    END_IF
																										 
															AuxOutputSelection.BagMadePlusLabelRequired:	//
																 									IF NOT printerDataReady AND state = HEAD_STATES.SealedAndSeparatedBag THEN
																										configOutput1Pulse.ManualOn();
																									END_IF
																									
																									IF printerDataReady OR HMIData.faultActive OR (releaseAndFeedSubState = RELEASE_FEED_STATES.FeedToOffset) THEN
																										configOutput1Pulse.ManualOff();
																									END_IF 
															AuxOutputSelection.BagsLow:				//
																									IF HMIData.bagLevelLow.active THEN
																										configOutput1Pulse.ManualOn();
																									ELSE
																										configOutput1Pulse.ManualOff();
																									END_IF											 
															
														END_CASE
															 
														CASE HMIData.auxIOConfig.cfgOutput2Selection OF
																 
															AuxOutputSelection.BagMade:				//
																 									IF state = HEAD_STATES.SealedAndSeparatedBag THEN
																										configOutput2Pulse.Trigger();
																									END_IF
																										 
															AuxOutputSelection.CycleComplete:		//
																 									IF state = HEAD_STATES.OpenedBag THEN
																										configOutput2Pulse.Trigger();
																									END_IF
																										 
															AuxOutputSelection.PrinterDataReady:	//
																 									IF printerDataReady THEN
																										configOutput2Pulse.ManualOn();
																									ELSE
																										configOutput2Pulse.ManualOff();
																									END_IF
																										 
															AuxOutputSelection.WaitingForPrinter:	// 
																 									IF releaseAndFeedSubState = RELEASE_FEED_STATES.WaitForPrinter THEN
																										configOutput2Pulse.ManualOn();
																									ELSE
																										configOutput2Pulse.ManualOff();	
																								    END_IF
																										 
															AuxOutputSelection.BagMadePlusLabelRequired:	//
																 									IF NOT printerDataReady AND state = HEAD_STATES.SealedAndSeparatedBag THEN
																										configOutput2Pulse.ManualOn();
																									END_IF
																									
																									IF printerDataReady OR HMIData.faultActive OR (releaseAndFeedSubState = RELEASE_FEED_STATES.FeedToOffset) THEN
																										configOutput2Pulse.ManualOff();
																									END_IF 
																										 
															AuxOutputSelection.BagsLow:				//
																									IF HMIData.bagLevelLow.active THEN
																										configOutput2Pulse.ManualOn();
																									ELSE
																										configOutput2Pulse.ManualOff();
																									END_IF	
														END_CASE
														
		 
END_CASE 
	 
// Pulse outputs that are temporary statuses (Cycle Complete) vs. held (Waiting for Printer) 
configOutput1Pulse(Q => oAuxConfigOut1);
configOutput2Pulse(Q => oAuxConfigOut2);
configOutput1Pulse.DwellSetting := 500;
configOutput2Pulse.DwellSetting := 500;
 // Filler and EZFeed conveyor setup
CASE HMIData.fillerFactorySelection OF
	FillerSelection.NotInstalled:					// No filler
		 											filler.enable := FALSE;
													filler.activateFiller := FALSE;	
													ezfeed.enable := FALSE;
													fillerModeCycleStartOnlyPulse.Reset();
													Infeed_Conveyor_IO.Enable := FALSE;
		 
	FillerSelection.StandardFiller:					// Only enable filler if Aux IO is enabled
		 											filler.enable := (HMIData.auxIOConfig.factorySelection = AuxiliaryIOSelection.AuxIOStandard);
													Infeed_Conveyor_IO.Enable := FALSE;
														 
	FillerSelection.EZFeed:							filler.enable := TRUE;
		 											ezfeed.enable := TRUE;
													Infeed_Conveyor_IO.Enable := TRUE;
													
		 											

END_CASE 
	 
ezfeed(
	enable:= , 
	baggerFaulted:= HMIData.faultActive, 
	enableEZFeed:= HMIData.fillerEnable, 
	continuousModeEnable:= HMIData.infeedConveyorRunningMode, 
	partsCountingModeEnable:= HMIData.infeedConveyorCountingMode, 
	flightPresentSensor:= iInfeedFlightSensor, 
	partPresentSensor:= , 
	waitingForFiller:= filler.waitingForFiller, 
	indexDwellSetting:= HMIData.infeedIndexDwellTimer, 
	flightTarget:= HMIData.infeedFlightCountTarget, 
	partsTarget:= HMIData.infeedPartsCountTarget, 
	emptyPartsWarningSetting:= HMIData.infeedEmptyPartsSetting, 
	restartFromEmptyParts:= HMIData.initiateCycle, 
	state=> , 
	runVFD=> oRunInfeedVFD, 
	flightCount=> HMIData.infeedFlightCountActual, 
	partsCount=> HMIData.infeedPartsCountActual, 
	emptyPartsWarningCount=> HMIData.infeedEmptyPartsActual, 
	emptyPartsWarning=> HMIData.infeedConveyorOutOfParts.active,
	EZFeedDone=> );

IF HMIData.fillerFactorySelection = FillerSelection.EZFeed THEN
	Infeed_Conveyor_IO.Enable := TRUE; 
	IF Infeed_Conveyor_IO.udiState <> 4  THEN 
		infeedConveyorIOCommFail.Trigger();
	END_IF
ELSE
	Infeed_Conveyor_IO.Enable := FALSE;
END_IF
	 
infeedConveyorVFDFaulted.faultTrigger := (HMIData.fillerFactorySelection = FillerSelection.EZFeed) AND NOT iInfeedVFDNotFaulted;
	
fillerModeCycleStartOnlyPulse.DwellSetting := 4000;
fillerModeCycleStartOnlyPulse(Q => HMIData.fillerModeCycleStartOnly.active);
filler(
	enable:= , 
	fillerTrigger:= iAuxFillerTrigger OR ezfeed.EZFeedDone,
	fillerOK:= iAuxFillerOK, 
	activateFiller:= HMIData.fillerEnable, 
	dropTime:= HMIData.fillerDropTime,
	state=> , 
	fillerModeActive=> , 
	waitingForFiller=> ,
	cycleBagRequest=> , 
	cycleBaggerToActivateFiller=> , 
	notReady=> );	 
IF filler.activateFiller AND NOT filler.cycleBaggerToActivateFiller.active THEN
	IF HMIData.initiateCycle OR startCycleReqFromPalmButtons THEN
		fillerModeCycleStartOnlyPulse.Trigger();
	END_IF
END_IF
	 

HMIData.packageEjectGuardRemoved.active :=  HMIData.packageEjectSelection = PackageEjectionSelection.LabelSideUp AND NOT iPackageEjectGuardClosed;
HMIData.loadPlateService.extendedFeedback := HMIData.rearLoadPlateService.extendedFeedback := iLoadPlateExtended;
HMIData.loadPlateService.retractedFeedback := HMIData.rearLoadPlateService.retractedFeedback := iLoadPlateRetracted;

rearLoadPlateRetract();
oLoadPlateRetract := rearLoadPlateRetract.Q;
oLoadPlateExtend := NOT oLoadPlateRetract;
loadPlateFaultTimer(
	enable:= , 
	extendCommand:= oLoadPlateExtend, 
	extendedInput:= iLoadPlateExtended, 
	retractCommand:= oLoadPlateRetract, 
	retractedInput:= iLoadPlateRetracted, 
	faultTime:= , 
	failToExtend=> loadPlateFaults.failedToLoad.faultTrigger, 
	failToRetract=> loadPlateFaults.failedToDischarge.faultTrigger);
rearLoadPlateFaultTimer(
	enable:= , 
	extendCommand:= oLoadPlateExtend, 
	extendedInput:= iLoadPlateExtended, 
	retractCommand:= oLoadPlateRetract, 
	retractedInput:= iLoadPlateRetracted, 
	faultTime:= , 
	failToExtend=> rearLoadPlateFaults.failedToLoad.faultTrigger, 
	failToRetract=> rearLoadPlateFaults.failedToDischarge.faultTrigger);

HMIData.forwardLoadPlateService.extendedFeedback := iFrontLoadPlateExtended;
HMIData.forwardLoadPlateService.retractedFeedback := iFrontLoadPlateRetracted;
forwardLoadPlateRetract.DwellSetting := TO_UINT(HMIData.loadPlateDwell * 1000);
forwardLoadPlateRetract.DelaySetting := TO_UINT(HMIData.loadPlateDelay * 1000);
forwardLoadPlateRetract();
oFrontLoadPlateToLoad := NOT forwardLoadPlateRetract.Q;
forwardLoadPlateFaultTimer(
	enable:= , 
	extendCommand:= NOT oFrontLoadPlateToLoad, 
	extendedInput:=iFrontLoadPlateExtended, 
	retractCommand:= oFrontLoadPlateToLoad, 
	retractedInput:= iFrontLoadPlateRetracted, 
	faultTime:= , 
	failToExtend=> forwardLoadPlateFaults.failedToLoad.faultTrigger, 
	failToRetract=> forwardLoadPlateFaults.failedToDischarge.faultTrigger);
		 
HMIData.loadShelfService.extendedFeedback := iLoadShelfExtended;
HMIData.loadShelfService.retractedFeedback := iLoadShelfRetracted;
loadShelfExtend.DwellSetting := TO_UINT(HMIData.loadPlateDwell * 1000);
loadShelfExtend.DelaySetting := TO_UINT(HMIData.loadPlateDelay * 1000);
loadShelfExtend();
oLoadShelfUp := NOT loadShelfExtend.Q;
loadShelfFaultTimer(
	enable:= , 
	extendCommand:= NOT oLoadShelfUp, 
	extendedInput:=iLoadShelfExtended, 
	retractCommand:= oLoadShelfUp, 
	retractedInput:= iLoadShelfRetracted, 
	faultTime:= , 
	failToExtend=> loadShelfFaults.failedToDischarge.faultTrigger, 
	failToRetract=> loadShelfFaults.failedToLoad.faultTrigger);
 
exitConveyorRun();
exitConveyorRun.DwellSetting := TO_UINT(HMIData.exitConveyorDwell * 1000);
exitConveyorJogONS(CLK := HMIData.exitConveyorJog);
oRunExitConveyor := exitConveyorRun.Q AND HMIData.integratedExitConveyorSelection = IntegratedConveyorSelection.RearExit;
	 
externalExitConveyorRun();
externalExitConveyorRun.DwellSetting := TO_UINT(HMIData.externalExitConveyorDwell * 1000);
externalExitConveyorJogONS(CLK := HMIData.externalExitConveyorJog);
oRunExternalExitConveyor := externalExitConveyorRun.Q AND HMIData.externalExitConveyorSelection <> ExteralConveyorSelection.NotInstalled;

bagOpenFingers(enable := HMIData.bofSelection <> BagOpenFingersSelection.NotInstalled,
				releaseOutput => oBOFUp,
		 		grabOutput => oBOFDown,
				rightFingerBagPresent := iRightFingerBagPresent,
				leftFingerBagPreset := iLefttFingerBagPresent,
				bagFailedToGrabBothFingersCount := Globals.bagFailedToGrabBothFingersCount,
				bagFailedToGrabLeftFingerCount := Globals.bagFailedToGrabLeftFingerCount,
				bagFailedToGrabRightFingerCount := Globals.bagFailedToGrabRightFingerCount,
				successfulBagOpenCount := Globals.successfulBagOpenCount);
					 
			



// Setup and run adjustable passthrough
//refIECObject := Pbar_ServoEIP;
pressureBarEndStopMotor(ptrEIPInputs := ADR(jawPasstrhoughMotorInputs),
                ptrEIPOutputs := ADR(jawPasstrhoughMotorOutputs),
                stepsPerInchSetpoint := Globals.STEPS_PER_INCH_SHOW_MOTOR,
				reversePolarity := TRUE,
				defaultCurrentSetpoint := 650,
				commFail := Pbar_ServoEIP.udiState <> 4,
				isHomable := TRUE);			
pressureBarEndStopMotor.Execute();

passthrough(pressureBarEndStopMotor := pressureBarEndStopMotor, 
			cumulativeChangeCount := Globals.passthroughChangeCount2, 
			cumulativeChangeDistance := Globals.passthroughChangeDistance2,
			jogInPB := HMIData.jogPassthroughForward,
			jogOutPB := HMIData.jogPassthroughReverse,
			passthroughPosition => HMIData.passthroughPosition);
passthrough.Mode := passthroughMode;


{endregion}
	 
hmiLight(lightOutput => oHMILight);
faultONS(CLK := HMIData.faultActive);

readyToRun := (motorizedSealFlatteners.Ready OR NOT motorizedSealFlatteners.enable) 
                AND (pressureBar.Ready OR NOT pressureBar.enable)
                AND (bagDelivery.Ready OR NOT bagDelivery.enable)
                AND (zebraPrinter.Ready OR NOT zebraPrinter.enable)
				AND (passthrough.Ready OR NOT passthrough.enable)
				AND murrIOBusNode.ok;
iPowerOffButtonONS(CLK := iPowerOffButton);

				
IF HMIData.makeReady OR iPowerOffButton THEN
	HMIData.ackAllFaults := TRUE;
	enable := TRUE;
	
	bagDropTimer.IN := FALSE;
	
	motorizedSealFlattenersMode := DEVICE_MODES.Auto;
	motorizedSealFlatteners.Reset();
	motorizedSealFlatteners.enable := HMIData.sealFlattenersSelection = SealFlattenerSelection.MotorizedSealFlatteners;
	IF motorizedSealFlatteners.sealFlattenersHorizontalAxisMotor.HomeRequired AND HMIData.sealFlattenersSelection = SealFlattenerSelection.MotorizedSealFlatteners THEN
		motorizedSealFlatteners.sealFlattenersHorizontalAxisMotor.HomeNow();
		motorizedSealFlatteners.sealFlattenersVerticalAxis.Retract();
	END_IF
	
	HMIData.bagOpenFeedNewBagCount := 0;
	bagOpenRetryCount := 0;
	
	HMIData.stopMachine := FALSE;
	
	electricPressureBarMode := DEVICE_MODES.Auto;
	pressureBar.Reset();
	pressureBar.enable := TRUE;
	//pressureBar.ExtendCylinderLowPressure();
	
	//HMIData.sealBarTemperatureSetting := 300;
	enableHeater := TRUE;
	
	bagDeliveryMode := DEVICE_MODES.Auto;
	bagDelivery.Reset();
	bagDelivery.enable := TRUE;
	//bagDelivery.bagFeedMasterMotor.SetRearMotorToTorqueMode();
	IF iPowerOffButtonONS.OSR THEN
		bagDelivery.AutoFeedToEye();
	END_IF
	bagOpened := FALSE;
	
	enableBatch := FALSE;
	batchCount := 0;
	
	//zebraPrinter.autoSendLabel := TRUE;
	printerMode := DEVICE_MODES.Auto;
	zebraPrinter.Reset();
	//zebraPrinter.enable := TRUE;
	
	IF iPowerOffButtonONS.OSR AND NOT bagDelivery.bagTensionFault.active THEN
		IF (HMIData.factoryTestMode AND (HMIData.bagsMade.count < 1000)) THEN
			HMIData.bagsMade.Clear();
		END_IF 
	END_IF  
	passthrough.Reset();
	pressureBarEndStopMotor.Reset();
	passthroughMode := DEVICE_MODES.Auto;
	passthrough.enable := TRUE;
	IF passthrough.homeRequired THEN
		homeJawPB := TRUE;
	ELSE
		pressureBar.ExtendCylinderLowPressure();
	END_IF
	oVacOn := FALSE;
	rearLoadPlateRetract.Reset();
	forwardLoadPlateRetract.Reset();
	loadShelfExtend.Reset();
	IBDRetractToDeflate.Reset();
	IBDRetractToEject.Reset();
	IBDCylinders.Extend();
	LPA.Reset();
	LPA.ManualOff();
	HPA.Reset();
	funnel.CloseNow();
	exitConveyorRun.Reset();
	externalExitConveyorRun.Reset();
	oSealBarExtend := FALSE;
	oSealBarRetract := TRUE;
	sealTimer.IN := FALSE;
	pressureBarCloseDelay.IN := FALSE;
	filler.Reset();
	configOutput1Pulse.Reset();
	configOutput2Pulse.Reset();
	configOutput1Pulse.ManualOff();
	configOutput2Pulse.ManualOff();
	fillerModeCycleStartOnlyPulse.Reset();
	barcodeVerifier.Reset();
	keyenceBCV.Reset();
	//HMIData.airFilterClean.SetCount(27336);
	//HMIData.driveRollerClean.SetCount(12041);
	//HMIData.printHeadClean.SetCount(3224);
	//HMIData.pressureBarGuideShaftGuides.SetCount(127888);
	
	//HMIData.bagLength := 23.5;
	//HMIData.bagWidth := 17.5;
	//HMIData.bagReverseSpeed := 3;
// 	HMIData.printLength := 8;
// 	HMIData.printOffset := 1;
// 	HMIData.printSpeed := 6;
// 	HMIData.bagForwardSpeed := 50;
	state := HEAD_STATES.Idle;
	reset();
	setPassthroughPB := FALSE;
	//homeJawPB := FALSE;
	HMIData.jobLoadRequired.active := TRUE;
	HMIData.makeReady := FALSE;
	bagDelivery.bagFeedRearMotor.SetRearMotorTorqueValue(TO_DINT(HMIDAta.bagTensionSetting * 100));
	hmiLight.TurnOff();
	
END_IF
IF enableONS.Q OR resetONS.Q THEN
    state := HEAD_STATES.Idle;
	sealAndSeparateSubState := SEAL_SEPARATE_STATES.Idle;
	releaseAndFeedSubState := RELEASE_FEED_STATES.Idle;
	openBagSubState := BAG_OPEN_ASSIST_STATES.Idle;
	finishCycleSubState := FINISH_CYCLE_STATES.Idle;
	motorizedSealFlatteners.Reset();
	pressureBar.Reset();
	bagDelivery.Reset();
	zebraPrinter.Reset();
	//pressureBar.ExtendCylinderLowPressure();
	bagDropTimer.IN := FALSE;
	_reset := FALSE;
	cycleTimer.IN := FALSE;
//	bagFailedToOpen := FALSE;
END_IF

{warning 'TODO: Put this inside the passtrough FB'}
IF passthrough.exhaustPressureBarRequest THEN
    pressureBar.ExhaustCylinder();
	IBDCylinders.Exhaust();
	IF NOT oPBar1Extend AND NOT oPBar1Retract THEN
		passthrough.AckRequest();
	END_IF
ELSIF passthrough.extendPressureBarRequest THEN
    pressureBar.ExtendCylinderLowPressure();
	IBDCylinders.Extend();
	IF oPBar1Extend AND oPBar1Retract THEN
		passthrough.AckRequest();
	END_IF
END_IF

IF HMIData.bagsMade.count >= 1000 THEN
	Globals.factoryTestComplete := TRUE;
END_IF

IF Globals.factoryTestComplete THEN
	HMIData.machineNotTested.active := FALSE;
ELSE
	HMIData.machineNotTested.active := TRUE;
END_IF

IF HMIData.factoryTestMode THEN
	HMIData.factoryTestModeActive.active := TRUE;
ELSE
	HMIData.factoryTestModeActive.active := FALSE;
END_IF

// Disable the printer on dry cycle because we dont't want to print on the platen roller               
IF Globals.enableDryCycle THEN
    zebraPrinter.enable := FALSE;
END_IF

// Send torque value to motor                 
rearMotorCommsReturned(CLK := bagDelivery.bagFeedRearMotor.commFail);
IF HMIData.jobLoaded OR rearMotorCommsReturned.Q THEN
	bagDelivery.bagFeedRearMotor.SetRearMotorTorqueValue((TO_DINT(HMIData.bagTensionSetting * 100)));
END_IF

// Clear batch count on batch enable
enableBatchONS(CLK := enableBatch);
IF enableBatchONS.Q THEN
    batchCount := 0;
END_IF

IF NOT enable OR NOT readyToRun OR faultONS.OSR THEN
    state := HEAD_STATES.Fault;
	enableBatch := FALSE;
	pressureBarEndStopMotor.Stop();
	cycleTimer.IN := FALSE;
END_IF
pressureBarCloseDelay(PT := TO_TIME(HMIData.pressureBarCloseDelay * 1000));
cycleTimer();
IF state <> HEAD_STATES.Idle AND HMIData.initiateCycle THEN
	HMIData.initiateCycle := FALSE;
END_IF
CASE state OF
    HEAD_STATES.Idle :                                // Start cycle if enabled
													
													
                                                    IF (startCycle AND (filler.cycleBaggerToActivateFiller.active OR NOT filler.activateFiller)
													OR (enableBatch AND (batchCount < batchSetting))
													OR (HMIData.factoryTestMode AND (HMIData.bagsMade.count < 1000)) AND factoryTestModeKeepCycling AND NOT LPA.Q
													OR startCycleReqFromPalmButtonsONS.OSR AND (filler.cycleBaggerToActivateFiller.active OR NOT filler.activateFiller)
													OR (HMIData.initiateCycle AND readyToRun) AND (filler.cycleBaggerToActivateFiller.active OR NOT filler.activateFiller)
													OR filler.cycleBagRequest) 
													AND NOT HMIData.faultActive 
													AND NOT HMIData.stopMachine 
													AND NOT HMIData.baggerInhibited.active
													AND NOT HMIData.sealBarNotAtTemperature.active
													AND NOT setPassthroughPB THEN
                                                        state := HEAD_STATES.SealAndSeparateBag;
                                                        startCycle := FALSE;
														
														cycleTimer.IN := TRUE;
                                                    END_IF
													IF NOT Globals.passthroughChangedFromJog AND HMIData.jobLoaded THEN
														HMIData.jobLoaded := FALSE;
													END_IF
                                                    IF (HMIData.passthroughSetting <> passthroughSettingLast) OR (Globals.passthroughChangedFromJog AND HMIData.jobLoaded) AND NOT pressureBarEndStopMotor.Faulted AND NOT pressureBarEndStopMotor.HomeRequired THEN
															setPassthroughPB := TRUE;
															Globals.passthroughChangedFromJog := FALSE;
															HMIData.jobLoaded := FALSE;
															passthroughSetting := HMIData.passthroughSetting;
															passthroughSettingLast := HMIData.passthroughSetting;
													END_IF
													
													IF (NOT pressureBarEndStopMotor.HomeRequired OR pressureBarEndStopMotor.Faulted)
														AND (NOT motorizedSealFlatteners.sealFlattenersHorizontalAxisMotor.homeRequiredIndication OR motorizedSealFlatteners.sealFlattenersHorizontalAxisMotor.Faulted)
														AND readyToRun 
														AND NOT HMIData.faultActive
													THEN
														hmiLight.TurnOn();
													END_IF
													
													
													IF HMIData.stopMachine THEN
														setPassthroughPB := FALSE;
														homeJawPB := FALSE;
														startCycle := FALSE;
														HMIData.initiateCycle := FALSE;
														factoryTestModeKeepCycling := FALSE;
														hmiLight.TurnOff();
													END_IF
													
													IF HMIData.sealBarNotAtTemperature.active THEN
														factoryTestModeKeepCycling := FALSE;
													END_IF
													
													IF bagOpened THEN
														IF NOT bagOpenFingers.CheckIfBagGrabbed(FALSE) THEN
															openedBagWasRemoved.Trigger();
															bagOpened := FALSE;
														END_IF
													END_IF
													
													{region:'Service'}
													IF setPassthroughPB AND NOT homeJawPB THEN
														hmiLight.BlinkSlow();
														state := HEAD_STATES.MovePassthrough;
													END_IF
													IF homeJawPB THEN
														hmiLight.BlinkSlow();
														state := HEAD_STATES.StartHoming;
													END_IF    
													
													IF HMIData.loadPlateService.retractCommand OR HMIData.rearLoadPlateService.retractCommand THEN
														rearLoadPlateRetract.ManualOn();
														HMIData.loadPlateService.retractCommand := FALSE;
														HMIData.rearLoadPlateService.retractCommand := FALSE;
													END_IF                                      
                                                    
													IF HMIData.loadPlateService.extendCommand OR HMIData.rearLoadPlateService.extendCommand THEN
														rearLoadPlateRetract.ManualOff();
														HMIData.loadPlateService.extendCommand := FALSE;
														HMIData.rearLoadPlateService.extendCommand := FALSE;
													END_IF
													
													IF HMIData.loadShelfService.retractCommand THEN
														loadShelfExtend.ManualOn();
														HMIData.loadShelfService.retractCommand := FALSE;
													END_IF                                      
                                                    
													IF HMIData.loadShelfService.extendCommand THEN
														loadShelfExtend.ManualOff();
														HMIData.loadShelfService.extendCommand := FALSE;
													END_IF	

													IF HMIData.forwardLoadPlateService.retractCommand THEN
														forwardLoadPlateRetract.ManualOn();
														HMIData.forwardLoadPlateService.retractCommand := FALSE;
													END_IF                                      
                                                    
													IF HMIData.forwardLoadPlateService.extendCommand THEN
														forwardLoadPlateRetract.ManualOff();
														HMIData.forwardLoadPlateService.extendCommand := FALSE;
													END_IF	 
													
													IF HMIData.IBDService.retractCommand THEN
														IBDCylinders.Retract();
														HMIData.IBDService.retractCommand := FALSE;
													END_IF                                      
                                                    
													IF HMIData.IBDService.extendCommand THEN
														IBDCylinders.Extend();
														HMIData.IBDService.extendCommand := FALSE;
													END_IF	
														 
													IF HMIData.funnelService.retractCommand THEN
														funnel.OpenNow();
														HMIData.funnelService.retractCommand := FALSE;
													END_IF                                      
                                                    
													IF HMIData.funnelService.extendCommand THEN
														funnel.CloseNow();
														HMIData.funnelService.extendCommand := FALSE;
													END_IF	
	 
													IF HMIData.lpaServicePulse THEN
														LPA.Trigger();
														HMIData.lpaServicePulse := FALSE;
													ELSIF HMIData.lpaServiceOn THEN
														LPA.ManualOn();
														HMIData.lpaServiceOn := FALSE;
													ELSIF HMIData.lpaServiceOff THEN
														LPA.ManualOff();
														HMIData.lpaServiceOff := FALSE;
													END_IF
													
													IF HMIData.vacuumServiceOn THEN
														oVacOn := TRUE;
														HMIData.vacuumServiceOn := FALSE;
													ELSIF HMIData.vacuumServiceOff THEN
														oVacOn := FALSE;
														HMIData.vacuumServiceOff := FALSE;
													END_IF
														 
															  
													IF HMIData.hpaServicePulse THEN
														hpa.Trigger();
														HMIData.hpaServicePulse := FALSE;
													ELSIF hpaServiceOnONS.OSR THEN
														HPA.ManualOn();
													ELSIF hpaServiceOnONS.OSF THEN
														HPA.ManualOff();
													END_IF
													
													IF HMIData.exitConveyorStartDwell THEN
														exitConveyorRun.Trigger();
														HMIData.exitConveyorStartDwell := FALSE;
													ELSIF HMIData.exitConveyorStart OR exitConveyorJogONS.OSR THEN
														exitConveyorRun.ManualOn();
														HMIData.exitConveyorStart := FALSE;
													ELSIF HMIData.exitConveyorStop OR exitConveyorJogONS.OSF THEN
														exitConveyorRun.ManualOff();
														HMIData.exitConveyorStop := FALSE;
													END_IF
													
													IF HMIData.externalExitConveyorStartDwell THEN
														externalExitConveyorRun.Trigger();
														HMIData.externalExitConveyorStartDwell := FALSE;
													ELSIF HMIData.externalExitConveyorStart OR externalExitConveyorJogONS.OSR THEN
														externalExitConveyorRun.ManualOn();
														HMIData.externalExitConveyorStart := FALSE;
													ELSIF HMIData.externalExitConveyorStop OR externalExitConveyorJogONS.OSF THEN
														externalExitConveyorRun.ManualOff();
														HMIData.externalExitConveyorStop := FALSE;
													END_IF
	 
													IF HMIData.sealBarServiceCycle THEN
														sealTimer.PT := TO_TIME(HMIData.sealBarDwell * 1000);
														sealTimer.IN := TRUE;
														IF NOT sealTimer.Q THEN
															oSealBarExtend := TRUE;
															oSealBarRetract := FALSE;
														ELSE 
															sealTimer.IN := FALSE;
															oSealBarExtend := FALSE;
															oSealBarRetract := TRUE;
															HMIData.sealBarCycles.Increment();
															HMIData.sealBarServiceCycle := FALSE;
														END_IF
													ELSIF HMIData.sealBarServiceExtend THEN
														oSealBarExtend := TRUE;
														oSealBarRetract := FALSE;
														HMIData.sealBarServiceExtend := FALSE;
													ELSIF HMIData.sealBarServiceRetract THEN
														oSealBarExtend := FALSE;
														oSealBarRetract := TRUE;
														HMIData.sealBarServiceRetract := FALSE;
													END_IF
														 
													IF HMIData.bagOpenFingersServiceGrab THEN
														bagOpenFingers.Grab();
														HMIData.bagOpenFingersServiceGrab := FALSE;
													ELSIF HMIData.bagOpenFingersServiceRelease THEN
														bagOpenFingers.Release();
														HMIData.bagOpenFingersServiceRelease := FALSE;
													END_IF
		  
													{endregion:'Service'}
                                                    
    HEAD_STATES.SealAndSeparateBag :                // Begin Seal and Separate State machine
													IF enableIBDDeflate THEN
														sealAndSeparateSubState := SEAL_SEPARATE_STATES.BringInIBD;
													ELSE
														sealAndSeparateSubState := SEAL_SEPARATE_STATES.WaitForJawCloseDelay;
													END_IF
													filler.BaggerCycleInitiated();
                                                    HMIData.inCycle := TRUE;
													HMIData.airFilterClean.Increment();
													HMIData.baggerCycles.Increment();
													IF funnel.enable THEN
														funnel.CloseNow();
													END_IF
													
                                                    state := HEAD_STATES.SealingAndSeparatingBag;
                                                    
                
    HEAD_STATES.SealingAndSeparatingBag :            IF sealAndSeparateSubState = SEAL_SEPARATE_STATES.Done THEN
                                                        state := HEAD_STATES.SealedAndSeparatedBag;
                                                        sealAndSeparateSubState := SEAL_SEPARATE_STATES.Idle;
                                                    END_IF    

    HEAD_STATES.SealedAndSeparatedBag :                state := HEAD_STATES.ReleaseAndFeedBag;                                    
                                                    
    HEAD_STATES.ReleaseAndFeedBag :                    // Open the jaw and release the bag
                                                    releaseAndFeedSubState := RELEASE_FEED_STATES.MoveJawOutAndDropBag;
                                                    state := HEAD_STATES.ReleasingAndFeedingBag;
                                                    
    HEAD_STATES.ReleasingAndFeedingBag :            // 
                                                    IF releaseAndFeedSubState = RELEASE_FEED_STATES.Done THEN
                                                        state := HEAD_STATES.ReleasedAndFedBag;
                                                        releaseAndFeedSubState := RELEASE_FEED_STATES.Idle;
                                                    END_IF
                                                    
    HEAD_STATES.ReleasedAndFedBag :                    // 
                                                    {warning 'TODO: change this counting logic to account for MSF'}
                                                    IF enableBatch THEN
                                                        batchCount := batchCount + 1;
                                                    END_IF
  
